gfCNCPoint2[22796] = {X 363.4255, Y 42.5965, Z -3.0000, A 0.000, B 0.000, C 0.000 }
gfCNCPoint2[22797] = {X 362.0806, Y 43.9848, Z -3.0000, A 0.000, B 0.000, C 0.000 }
gfCNCPoint2[22798] = {X 360.6191, Y 45.2499, Z -3.0000, A 0.000, B 0.000, C 0.000 }
gfCNCPoint2[22799] = {X 359.0523, Y 46.3820, Z -3.0000, A 0.000, B 0.000, C 0.000 }
gfCNCPoint2[22800] = {X 357.3923, Y 47.3724, Z -3.0000, A 0.000, B 0.000, C 0.000 }
gfCNCPoint2[22801] = {X 355.4454, Y 48.2565, Z -3.0000, A 0.000, B 0.000, C 0.000 }
gfCNCPoint2[22802] = {X 353.4232, Y 48.9515, Z -3.0000, A 0.000, B 0.000, C 0.000 }
gfCNCPoint2[22803] = {X 351.3441, Y 49.4512, Z -3.0000, A 0.000, B 0.000, C 0.000 }
gfCNCPoint2[22804] = {X 349.2270, Y 49.7510, Z -3.0000, A 0.000, B 0.000, C 0.000 }
gfCNCPoint2[22805] = {X 347.0909, Y 49.8483, Z -3.0000, A 0.000, B 0.000, C 0.000 }
gfCNCPoint2[22806] = {X 345.0381, Y 49.8138, Z -3.0000, A 0.000, B 0.000, C 0.000 }
gfCNCPoint2[22807] = {X 342.9961, Y 49.6015, Z -3.0000, A 0.000, B 0.000, C 0.000 }
gfCNCPoint2[22808] = {X 340.9802, Y 49.2128, Z -3.0000, A 0.000, B 0.000, C 0.000 }
gfCNCPoint2[22809] = {X 339.0056, Y 48.6507, Z -3.0000, A 0.000, B 0.000, C 0.000 }
gfCNCPoint2[22810] = {X 337.0871, Y 47.9195, Z -3.0000, A 0.000, B 0.000, C 0.000 }
gfCNCPoint2[22811] = {X 335.2394, Y 47.0246, Z -3.0000, A 0.000, B 0.000, C 0.000 }
gfCNCPoint2[22812] = {X 333.6461, Y 46.0400, Z -3.0000, A 0.000, B 0.000, C 0.000 }
gfCNCPoint2[22813] = {X 332.1356, Y 44.9327, Z -3.0000, A 0.000, B 0.000, C 0.000 }
gfCNCPoint2[22814] = {X 330.7173, Y 43.7094, Z -3.0000, A 0.000, B 0.000, C 0.000 }
gfCNCPoint2[22815] = {X 329.7931, Y 43.7230, Z -3.0000, A 0.000, B 0.000, C 0.000 }
gfCNCPoint2[22816] = {X 328.8887, Y 43.5322, Z -3.0000, A 0.000, B 0.000, C 0.000 }
gfCNCPoint2[22817] = {X 328.0488, Y 43.1465, Z -3.0000, A 0.000, B 0.000, C 0.000 }
gfCNCPoint2[22818] = {X 327.3148, Y 42.5847, Z -3.0000, A 0.000, B 0.000, C 0.000 }
gfCNCPoint2[22819] = {X 326.6925, Y 41.9780, Z -3.0000, A 0.000, B 0.000, C 0.000 }
gfCNCPoint2[22820] = {X 326.0873, Y 41.2331, Z -3.0000, A 0.000, B 0.000, C 0.000 }
gfCNCPoint2[22821] = {X 325.6690, Y 40.3693, Z -3.0000, A 0.000, B 0.000, C 0.000 }
gfCNCPoint2[22822] = {X 325.4597, Y 39.4326, Z -3.0000, A 0.000, B 0.000, C 0.000 }
gfCNCPoint2[22823] = {X 325.4707, Y 38.4730, Z -3.0000, A 0.000, B 0.000, C 0.000 }
gfCNCPoint2[22824] = {X 325.7013, Y 37.5413, Z -3.0000, A 0.000, B 0.000, C 0.000 }
gfCNCPoint2[22825] = {X 326.1392, Y 36.6874, Z -3.0000, A 0.000, B 0.000, C 0.000 }
gfCNCPoint2[22826] = {X 330.3725, Y 30.3577, Z -3.0000, A 0.000, B 0.000, C 0.000 }
gfCNCPoint2[22827] = {X 330.9516, Y 29.6673, Z -3.0000, A 0.000, B 0.000, C 0.000 }
gfCNCPoint2[22828] = {X 331.6658, Y 29.1179, Z -3.0000, A 0.000, B 0.000, C 0.000 }
gfCNCPoint2[22829] = {X 332.4815, Y 28.7351, Z -3.0000, A 0.000, B 0.000, C 0.000 }
gfCNCPoint2[22830] = {X 333.3606, Y 28.5370, Z -3.0000, A 0.000, B 0.000, C 0.000 }
gfCNCPoint2[22831] = {X 334.2616, Y 28.5327, Z -3.0000, A 0.000, B 0.000, C 0.000 }
gfCNCPoint2[22832] = {X 335.1425, Y 28.7226, Z -3.0000, A 0.000, B 0.000, C 0.000 }
gfCNCPoint2[22833] = {X 335.9617, Y 29.0978, Z -3.0000, A 0.000, B 0.000, C 0.000 }
gfCNCPoint2[22834] = {X 336.6810, Y 29.6405, Z -3.0000, A 0.000, B 0.000, C 0.000 }
gfCNCPoint2[22835] = {X 337.3163, Y 30.2523, Z -3.0000, A 0.000, B 0.000, C 0.000 }
gfCNCPoint2[22836] = {X 337.8308, Y 30.8659, Z -3.0000, A 0.000, B 0.000, C 0.000 }
gfCNCPoint2[22837] = {X 338.2182, Y 31.5666, Z -3.0000, A 0.000, B 0.000, C 0.000 }
gfCNCPoint2[22838] = {X 338.4642, Y 32.3286, Z -3.0000, A 0.000, B 0.000, C 0.000 }
gfCNCPoint2[22839] = {X 338.5597, Y 33.1236, Z -3.0000, A 0.000, B 0.000, C 0.000 }
gfCNCPoint2[22840] = {X 338.5011, Y 33.9222, Z -3.0000, A 0.000, B 0.000, C 0.000 }
gfCNCPoint2[22841] = {X 339.2995, Y 34.6500, Z -3.0000, A 0.000, B 0.000, C 0.000 }
gfCNCPoint2[22842] = {X 340.1353, Y 35.3347, Z -3.0000, A 0.000, B 0.000, C 0.000 }
gfCNCPoint2[22843] = {X 341.4519, Y 36.1996, Z -3.0000, A 0.000, B 0.000, C 0.000 }
gfCNCPoint2[22844] = {X 342.8804, Y 36.8633, Z -3.0000, A 0.000, B 0.000, C 0.000 }
gfCNCPoint2[22845] = {X 344.3905, Y 37.3116, Z -3.0000, A 0.000, B 0.000, C 0.000 }
gfCNCPoint2[22846] = {X 345.9498, Y 37.5350, Z -3.0000, A 0.000, B 0.000, C 0.000 }
gfCNCPoint2[22847] = {X 347.5251, Y 37.5286, Z -3.0000, A 0.000, B 0.000, C 0.000 }
gfCNCPoint2[22848] = {X 348.7008, Y 37.3905, Z -3.0000, A 0.000, B 0.000, C 0.000 }
gfCNCPoint2[22849] = {X 349.8485, Y 37.1001, Z -3.0000, A 0.000, B 0.000, C 0.000 }
gfCNCPoint2[22850] = {X 350.9485, Y 36.6625, Z -3.0000, A 0.000, B 0.000, C 0.000 }
gfCNCPoint2[22851] = {X 351.9820, Y 36.0851, Z -3.0000, A 0.000, B 0.000, C 0.000 }
gfCNCPoint2[22852] = {X 352.9314, Y 35.3779, Z -3.0000, A 0.000, B 0.000, C 0.000 }
gfCNCPoint2[22853] = {X 354.1005, Y 34.2424, Z -3.0000, A 0.000, B 0.000, C 0.000 }
gfCNCPoint2[22854] = {X 355.1123, Y 32.9647, Z -3.0000, A 0.000, B 0.000, C 0.000 }
gfCNCPoint2[22855] = {X 355.9496, Y 31.5665, Z -3.0000, A 0.000, B 0.000, C 0.000 }
gfCNCPoint2[22856] = {X 356.5983, Y 30.0713, Z -3.0000, A 0.000, B 0.000, C 0.000 }
gfCNCPoint2[22857] = {X 357.0473, Y 28.5046, Z -3.0000, A 0.000, B 0.000, C 0.000 }
gfCNCPoint2[22858] = {X 357.3230, Y 26.8012, Z -3.0000, A 0.000, B 0.000, C 0.000 }
gfCNCPoint2[22859] = {X 357.4354, Y 25.0793, Z -3.0000, A 0.000, B 0.000, C 0.000 }
gfCNCPoint2[22860] = {X 357.3833, Y 23.3545, Z -3.0000, A 0.000, B 0.000, C 0.000 }
gfCNCPoint2[22861] = {X 357.1672, Y 21.6425, Z -3.0000, A 0.000, B 0.000, C 0.000 }
gfCNCPoint2[22862] = {X 356.8264, Y 20.1740, Z -3.0000, A 0.000, B 0.000, C 0.000 }
gfCNCPoint2[22863] = {X 356.3065, Y 18.7588, Z -3.0000, A 0.000, B 0.000, C 0.000 }
gfCNCPoint2[22864] = {X 355.6155, Y 17.4189, Z -3.0000, A 0.000, B 0.000, C 0.000 }
gfCNCPoint2[22865] = {X 354.7641, Y 16.1748, Z -3.0000, A 0.000, B 0.000, C 0.000 }
gfCNCPoint2[22866] = {X 353.8628, Y 15.1697, Z -3.0000, A 0.000, B 0.000, C 0.000 }
gfCNCPoint2[22867] = {X 352.8268, Y 14.3041, Z -3.0000, A 0.000, B 0.000, C 0.000 }
gfCNCPoint2[22868] = {X 351.6776, Y 13.5959, Z -3.0000, A 0.000, B 0.000, C 0.000 }
gfCNCPoint2[22869] = {X 350.4387, Y 13.0595, Z -3.0000, A 0.000, B 0.000, C 0.000 }
gfCNCPoint2[22870] = {X 349.1358, Y 12.7062, Z -3.0000, A 0.000, B 0.000, C 0.000 }
gfCNCPoint2[22871] = {X 347.5974, Y 12.5009, Z -3.0000, A 0.000, B 0.000, C 0.000 }
gfCNCPoint2[22872] = {X 346.0456, Y 12.4729, Z -3.0000, A 0.000, B 0.000, C 0.000 }
gfCNCPoint2[22873] = {X 344.5007, Y 12.6227, Z -3.0000, A 0.000, B 0.000, C 0.000 }
gfCNCPoint2[22874] = {X 342.9832, Y 12.9482, Z -3.0000, A 0.000, B 0.000, C 0.000 }
gfCNCPoint2[22875] = {X 341.5129, Y 13.4452, Z -3.0000, A 0.000, B 0.000, C 0.000 }
gfCNCPoint2[22876] = {X 340.1091, Y 14.1071, Z -3.0000, A 0.000, B 0.000, C 0.000 }
gfCNCPoint2[22877] = {X 338.7902, Y 14.9254, Z -3.0000, A 0.000, B 0.000, C 0.000 }
gfCNCPoint2[22878] = {X 338.7680, Y 15.7568, Z -3.0000, A 0.000, B 0.000, C 0.000 }
gfCNCPoint2[22879] = {X 338.5809, Y 16.5673, Z -3.0000, A 0.000, B 0.000, C 0.000 }
gfCNCPoint2[22880] = {X 338.2362, Y 17.3243, Z -3.0000, A 0.000, B 0.000, C 0.000 }
gfCNCPoint2[22881] = {X 337.7479, Y 17.9976, Z -3.0000, A 0.000, B 0.000, C 0.000 }
gfCNCPoint2[22882] = {X 337.1353, Y 18.5603, Z -3.0000, A 0.000, B 0.000, C 0.000 }
gfCNCPoint2[22883] = {X 336.4209, Y 19.0861, Z -3.0000, A 0.000, B 0.000, C 0.000 }
gfCNCPoint2[22884] = {X 335.6353, Y 19.5283, Z -3.0000, A 0.000, B 0.000, C 0.000 }
gfCNCPoint2[22885] = {X 334.7729, Y 19.7908, Z -3.0000, A 0.000, B 0.000, C 0.000 }
gfCNCPoint2[22886] = {X 333.8742, Y 19.8614, Z -3.0000, A 0.000, B 0.000, C 0.000 }
gfCNCPoint2[22887] = {X 332.9814, Y 19.7367, Z -3.0000, A 0.000, B 0.000, C 0.000 }
gfCNCPoint2[22888] = {X 332.1364, Y 19.4226, Z -3.0000, A 0.000, B 0.000, C 0.000 }
gfCNCPoint2[22889] = {X 331.3789, Y 18.9339, Z -3.0000, A 0.000, B 0.000, C 0.000 }
gfCNCPoint2[22890] = {X 330.7445, Y 18.2934, Z -3.0000, A 0.000, B 0.000, C 0.000 }
gfCNCPoint2[22891] = {X 330.2630, Y 17.5314, Z -3.0000, A 0.000, B 0.000, C 0.000 }
gfCNCPoint2[22892] = {X 326.7381, Y 10.2803, Z -3.0000, A 0.000, B 0.000, C 0.000 }
gfCNCPoint2[22893] = {X 326.4156, Y 9.3505, Z -3.0000, A 0.000, B 0.000, C 0.000 }
gfCNCPoint2[22894] = {X 326.3205, Y 8.3711, Z -3.0000, A 0.000, B 0.000, C 0.000 }
gfCNCPoint2[22895] = {X 326.4581, Y 7.3967, Z -3.0000, A 0.000, B 0.000, C 0.000 }
gfCNCPoint2[22896] = {X 326.8207, Y 6.4819, Z -3.0000, A 0.000, B 0.000, C 0.000 }
gfCNCPoint2[22897] = {X 327.3881, Y 5.6778, Z -3.0000, A 0.000, B 0.000, C 0.000 }
gfCNCPoint2[22898] = {X 328.1285, Y 5.0296, Z -3.0000, A 0.000, B 0.000, C 0.000 }
gfCNCPoint2[22899] = {X 328.7983, Y 4.5709, Z -3.0000, A 0.000, B 0.000, C 0.000 }
gfCNCPoint2[22900] = {X 329.6633, Y 4.1255, Z -3.0000, A 0.000, B 0.000, C 0.000 }
gfCNCPoint2[22901] = {X 330.6082, Y 3.8933, Z -3.0000, A 0.000, B 0.000, C 0.000 }
gfCNCPoint2[22902] = {X 331.5811, Y 3.8868, Z -3.0000, A 0.000, B 0.000, C 0.000 }
gfCNCPoint2[22903] = {X 332.5290, Y 4.1066, Z -3.0000, A 0.000, B 0.000, C 0.000 }
gfCNCPoint2[22904] = {X 334.0387, Y 3.2602, Z -3.0000, A 0.000, B 0.000, C 0.000 }
gfCNCPoint2[22905] = {X 335.5974, Y 2.5081, Z -3.0000, A 0.000, B 0.000, C 0.000 }
gfCNCPoint2[22906] = {X 337.7207, Y 1.6466, Z -3.0000, A 0.000, B 0.000, C 0.000 }
gfCNCPoint2[22907] = {X 339.9113, Y 0.9746, Z -3.0000, A 0.000, B 0.000, C 0.000 }
gfCNCPoint2[22908] = {X 342.1523, Y 0.4972, Z -3.0000, A 0.000, B 0.000, C 0.000 }
gfCNCPoint2[22909] = {X 344.4266, Y 0.2179, Z -3.0000, A 0.000, B 0.000, C 0.000 }
gfCNCPoint2[22910] = {X 346.7166, Y 0.1391, Z -3.0000, A 0.000, B 0.000, C 0.000 }
gfCNCPoint2[22911] = {X 349.0046, Y 0.2612, Z -3.0000, A 0.000, B 0.000, C 0.000 }
gfCNCPoint2[22912] = {X 351.2732, Y 0.5834, Z -3.0000, A 0.000, B 0.000, C 0.000 }
gfCNCPoint2[22913] = {X 351.5567, Y 0.6360, Z -3.0000, A 0.000, B 0.000, C 0.000 }
gfCNCPoint2[22914] = {X 352.2862, Y -3.2969, Z -3.0000, A 0.000, B 0.000, C 0.000 }
gfCNCPoint2[22915] = {X 351.5421, Y 0.7147, Z -3.0000, A 0.000, B 0.000, C 0.000 }
gfCNCPoint2[22916] = {X 351.8236, Y 0.7669, Z -3.0000, A 0.000, B 0.000, C 0.000 }
gfCNCPoint2[22917] = {X 353.7359, Y 1.2474, Z -3.0000, A 0.000, B 0.000, C 0.000 }
gfCNCPoint2[22918] = {X 355.5941, Y 1.9070, Z -3.0000, A 0.000, B 0.000, C 0.000 }
gfCNCPoint2[22919] = {X 357.3815, Y 2.7397, Z -3.0000, A 0.000, B 0.000, C 0.000 }
gfCNCPoint2[22920] = {X 359.0818, Y 3.7380, Z -3.0000, A 0.000, B 0.000, C 0.000 }
gfCNCPoint2[22921] = {X 360.6799, Y 4.8930, Z -3.0000, A 0.000, B 0.000, C 0.000 }
gfCNCPoint2[22922] = {X 362.1614, Y 6.1942, Z -3.0000, A 0.000, B 0.000, C 0.000 }
gfCNCPoint2[22923] = {X 363.5129, Y 7.6299, Z -3.0000, A 0.000, B 0.000, C 0.000 }
gfCNCPoint2[22924] = {X 364.9659, Y 9.5050, Z -3.0000, A 0.000, B 0.000, C 0.000 }
gfCNCPoint2[22925] = {X 366.2305, Y 11.5119, Z -3.0000, A 0.000, B 0.000, C 0.000 }
gfCNCPoint2[22926] = {X 367.2950, Y 13.6318, Z -3.0000, A 0.000, B 0.000, C 0.000 }
gfCNCPoint2[22927] = {X 368.1493, Y 15.8448, Z -3.0000, A 0.000, B 0.000, C 0.000 }
gfCNCPoint2[22928] = {X 368.7853, Y 18.1301, Z -3.0000, A 0.000, B 0.000, C 0.000 }
gfCNCPoint2[22929] = {X 369.2628, Y 20.7447, Z -3.0000, A 0.000, B 0.000, C 0.000 }
gfCNCPoint2[22930] = {X 369.5173, Y 23.3903, Z -3.0000, A 0.000, B 0.000, C 0.000 }
gfCNCPoint2[22931] = {X 369.5471, Y 26.0480, Z -3.0000, A 0.000, B 0.000, C 0.000 }
gfCNCPoint2[22932] = {X 369.3519, Y 28.6987, Z -3.0000, A 0.000, B 0.000, C 0.000 }
gfCNCPoint2[22933] = {X 368.9331, Y 31.3234, Z -3.0000, A 0.000, B 0.000, C 0.000 }
gfCNCPoint2[22934] = {X 368.4143, Y 33.4074, Z -3.0000, A 0.000, B 0.000, C 0.000 }
gfCNCPoint2[22935] = {X 367.7134, Y 35.4375, Z -3.0000, A 0.000, B 0.000, C 0.000 }
gfCNCPoint2[22936] = {X 366.8358, Y 37.3977, Z -3.0000, A 0.000, B 0.000, C 0.000 }
gfCNCPoint2[22937] = {X 365.7884, Y 39.2726, Z -3.0000, A 0.000, B 0.000, C 0.000 }
gfCNCPoint2[22938] = {X 364.5794, Y 41.0477, Z -3.0000, A 0.000, B 0.000, C 0.000 }
gfCNCPoint2[22939] = {X 363.3659, Y 42.5431, Z -3.0000, A 0.000, B 0.000, C 0.000 }
gfCNCPoint2[22940] = {X 362.0260, Y 43.9264, Z -3.0000, A 0.000, B 0.000, C 0.000 }
gfCNCPoint2[22941] = {X 360.5699, Y 45.1869, Z -3.0000, A 0.000, B 0.000, C 0.000 }
gfCNCPoint2[22942] = {X 359.0089, Y 46.3148, Z -3.0000, A 0.000, B 0.000, C 0.000 }
gfCNCPoint2[22943] = {X 357.3551, Y 47.3015, Z -3.0000, A 0.000, B 0.000, C 0.000 }
gfCNCPoint2[22944] = {X 355.4150, Y 48.1825, Z -3.0000, A 0.000, B 0.000, C 0.000 }
gfCNCPoint2[22945] = {X 353.3999, Y 48.8750, Z -3.0000, A 0.000, B 0.000, C 0.000 }
gfCNCPoint2[22946] = {X 351.3281, Y 49.3728, Z -3.0000, A 0.000, B 0.000, C 0.000 }
gfCNCPoint2[22947] = {X 349.2184, Y 49.6715, Z -3.0000, A 0.000, B 0.000, C 0.000 }
gfCNCPoint2[22948] = {X 347.0899, Y 49.7683, Z -3.0000, A 0.000, B 0.000, C 0.000 }
gfCNCPoint2[22949] = {X 345.0440, Y 49.7340, Z -3.0000, A 0.000, B 0.000, C 0.000 }
gfCNCPoint2[22950] = {X 343.0088, Y 49.5225, Z -3.0000, A 0.000, B 0.000, C 0.000 }
gfCNCPoint2[22951] = {X 340.9996, Y 49.1352, Z -3.0000, A 0.000, B 0.000, C 0.000 }
gfCNCPoint2[22952] = {X 339.0316, Y 48.5751, Z -3.0000, A 0.000, B 0.000, C 0.000 }
gfCNCPoint2[22953] = {X 337.1196, Y 47.8464, Z -3.0000, A 0.000, B 0.000, C 0.000 }
gfCNCPoint2[22954] = {X 335.2780, Y 46.9545, Z -3.0000, A 0.000, B 0.000, C 0.000 }
gfCNCPoint2[22955] = {X 333.6799, Y 45.9664, Z -3.0000, A 0.000, B 0.000, C 0.000 }
gfCNCPoint2[22956] = {X 332.1655, Y 44.8542, Z -3.0000, A 0.000, B 0.000, C 0.000 }
gfCNCPoint2[22957] = {X 330.7443, Y 43.6252, Z -3.0000, A 0.000, B 0.000, C 0.000 }
gfCNCPoint2[22958] = {X 329.8287, Y 43.6460, Z -3.0000, A 0.000, B 0.000, C 0.000 }
gfCNCPoint2[22959] = {X 328.9316, Y 43.4621, Z -3.0000, A 0.000, B 0.000, C 0.000 }
gfCNCPoint2[22960] = {X 328.0980, Y 43.0827, Z -3.0000, A 0.000, B 0.000, C 0.000 }
gfCNCPoint2[22961] = {X 327.3701, Y 42.5270, Z -3.0000, A 0.000, B 0.000, C 0.000 }
gfCNCPoint2[22962] = {X 326.7483, Y 41.9207, Z -3.0000, A 0.000, B 0.000, C 0.000 }
gfCNCPoint2[22963] = {X 326.1548, Y 41.1901, Z -3.0000, A 0.000, B 0.000, C 0.000 }
gfCNCPoint2[22964] = {X 325.7445, Y 40.3430, Z -3.0000, A 0.000, B 0.000, C 0.000 }
gfCNCPoint2[22965] = {X 325.5393, Y 39.4243, Z -3.0000, A 0.000, B 0.000, C 0.000 }
gfCNCPoint2[22966] = {X 325.5500, Y 38.4831, Z -3.0000, A 0.000, B 0.000, C 0.000 }
gfCNCPoint2[22967] = {X 325.7762, Y 37.5694, Z -3.0000, A 0.000, B 0.000, C 0.000 }
gfCNCPoint2[22968] = {X 326.2057, Y 36.7318, Z -3.0000, A 0.000, B 0.000, C 0.000 }
gfCNCPoint2[22969] = {X 330.4390, Y 30.4021, Z -3.0000, A 0.000, B 0.000, C 0.000 }
gfCNCPoint2[22970] = {X 331.0069, Y 29.7251, Z -3.0000, A 0.000, B 0.000, C 0.000 }
gfCNCPoint2[22971] = {X 331.7073, Y 29.1862, Z -3.0000, A 0.000, B 0.000, C 0.000 }
gfCNCPoint2[22972] = {X 332.5073, Y 28.8108, Z -3.0000, A 0.000, B 0.000, C 0.000 }
gfCNCPoint2[22973] = {X 333.3694, Y 28.6165, Z -3.0000, A 0.000, B 0.000, C 0.000 }
gfCNCPoint2[22974] = {X 334.2530, Y 28.6123, Z -3.0000, A 0.000, B 0.000, C 0.000 }
gfCNCPoint2[22975] = {X 335.1169, Y 28.7985, Z -3.0000, A 0.000, B 0.000, C 0.000 }
gfCNCPoint2[22976] = {X 335.9204, Y 29.1663, Z -3.0000, A 0.000, B 0.000, C 0.000 }
gfCNCPoint2[22977] = {X 336.6259, Y 29.6985, Z -3.0000, A 0.000, B 0.000, C 0.000 }
gfCNCPoint2[22978] = {X 337.2602, Y 30.3094, Z -3.0000, A 0.000, B 0.000, C 0.000 }
gfCNCPoint2[22979] = {X 337.7696, Y 30.9181, Z -3.0000, A 0.000, B 0.000, C 0.000 }
gfCNCPoint2[22980] = {X 338.1515, Y 31.6139, Z -3.0000, A 0.000, B 0.000, C 0.000 }
gfCNCPoint2[22981] = {X 338.3914, Y 32.3705, Z -3.0000, A 0.000, B 0.000, C 0.000 }
gfCNCPoint2[22982] = {X 338.4804, Y 33.1593, Z -3.0000, A 0.000, B 0.000, C 0.000 }
gfCNCPoint2[22983] = {X 338.4149, Y 33.9503, Z -3.0000, A 0.000, B 0.000, C 0.000 }
gfCNCPoint2[22984] = {X 339.2312, Y 34.6967, Z -3.0000, A 0.000, B 0.000, C 0.000 }
gfCNCPoint2[22985] = {X 340.0864, Y 35.3980, Z -3.0000, A 0.000, B 0.000, C 0.000 }
gfCNCPoint2[22986] = {X 341.4126, Y 36.2693, Z -3.0000, A 0.000, B 0.000, C 0.000 }
gfCNCPoint2[22987] = {X 342.8516, Y 36.9379, Z -3.0000, A 0.000, B 0.000, C 0.000 }
gfCNCPoint2[22988] = {X 344.3727, Y 37.3896, Z -3.0000, A 0.000, B 0.000, C 0.000 }
gfCNCPoint2[22989] = {X 345.9434, Y 37.6147, Z -3.0000, A 0.000, B 0.000, C 0.000 }
gfCNCPoint2[22990] = {X 347.5302, Y 37.6085, Z -3.0000, A 0.000, B 0.000, C 0.000 }
gfCNCPoint2[22991] = {X 348.7161, Y 37.4690, Z -3.0000, A 0.000, B 0.000, C 0.000 }
gfCNCPoint2[22992] = {X 349.8737, Y 37.1760, Z -3.0000, A 0.000, B 0.000, C 0.000 }
gfCNCPoint2[22993] = {X 350.9832, Y 36.7345, Z -3.0000, A 0.000, B 0.000, C 0.000 }
gfCNCPoint2[22994] = {X 352.0257, Y 36.1521, Z -3.0000, A 0.000, B 0.000, C 0.000 }
gfCNCPoint2[22995] = {X 352.9832, Y 35.4388, Z -3.0000, A 0.000, B 0.000, C 0.000 }
gfCNCPoint2[22996] = {X 354.1599, Y 34.2960, Z -3.0000, A 0.000, B 0.000, C 0.000 }
gfCNCPoint2[22997] = {X 355.1782, Y 33.0101, Z -3.0000, A 0.000, B 0.000, C 0.000 }
gfCNCPoint2[22998] = {X 356.0208, Y 31.6029, Z -3.0000, A 0.000, B 0.000, C 0.000 }
gfCNCPoint2[22999] = {X 356.6736, Y 30.0982, Z -3.0000, A 0.000, B 0.000, C 0.000 }
gfCNCPoint2[23000] = {X 357.1255, Y 28.5214, Z -3.0000, A 0.000, B 0.000, C 0.000 }
gfCNCPoint2[23001] = {X 357.4025, Y 26.8104, Z -3.0000, A 0.000, B 0.000, C 0.000 }
gfCNCPoint2[23002] = {X 357.5154, Y 25.0808, Z -3.0000, A 0.000, B 0.000, C 0.000 }
gfCNCPoint2[23003] = {X 357.4630, Y 23.3484, Z -3.0000, A 0.000, B 0.000, C 0.000 }
gfCNCPoint2[23004] = {X 357.2460, Y 21.6288, Z -3.0000, A 0.000, B 0.000, C 0.000 }
gfCNCPoint2[23005] = {X 356.9029, Y 20.1507, Z -3.0000, A 0.000, B 0.000, C 0.000 }
gfCNCPoint2[23006] = {X 356.3797, Y 18.7264, Z -3.0000, A 0.000, B 0.000, C 0.000 }
gfCNCPoint2[23007] = {X 355.6842, Y 17.3778, Z -3.0000, A 0.000, B 0.000, C 0.000 }
gfCNCPoint2[23008] = {X 354.8272, Y 16.1256, Z -3.0000, A 0.000, B 0.000, C 0.000 }
gfCNCPoint2[23009] = {X 353.9182, Y 15.1120, Z -3.0000, A 0.000, B 0.000, C 0.000 }
gfCNCPoint2[23010] = {X 352.8735, Y 14.2391, Z -3.0000, A 0.000, B 0.000, C 0.000 }
gfCNCPoint2[23011] = {X 351.7144, Y 13.5249, Z -3.0000, A 0.000, B 0.000, C 0.000 }
gfCNCPoint2[23012] = {X 350.4650, Y 12.9840, Z -3.0000, A 0.000, B 0.000, C 0.000 }
gfCNCPoint2[23013] = {X 349.1511, Y 12.6277, Z -3.0000, A 0.000, B 0.000, C 0.000 }
gfCNCPoint2[23014] = {X 347.5971, Y 12.4206, Z -3.0000, A 0.000, B 0.000, C 0.000 }
gfCNCPoint2[23015] = {X 346.0297, Y 12.3935, Z -3.0000, A 0.000, B 0.000, C 0.000 }
gfCNCPoint2[23016] = {X 344.4695, Y 12.5466, Z -3.0000, A 0.000, B 0.000, C 0.000 }
gfCNCPoint2[23017] = {X 342.9373, Y 12.8779, Z -3.0000, A 0.000, B 0.000, C 0.000 }
gfCNCPoint2[23018] = {X 341.4532, Y 13.3830, Z -3.0000, A 0.000, B 0.000, C 0.000 }
gfCNCPoint2[23019] = {X 340.0371, Y 14.0553, Z -3.0000, A 0.000, B 0.000, C 0.000 }
gfCNCPoint2[23020] = {X 338.7075, Y 14.8858, Z -3.0000, A 0.000, B 0.000, C 0.000 }
gfCNCPoint2[23021] = {X 338.7152, Y 15.0050, Z -3.0000, A 0.000, B 0.000, C 0.000 }
gfCNCPoint2[23022] = {X 338.6808, Y 15.8053, Z -3.0000, A 0.000, B 0.000, C 0.000 }
gfCNCPoint2[23023] = {X 338.4907, Y 16.5835, Z -3.0000, A 0.000, B 0.000, C 0.000 }
gfCNCPoint2[23024] = {X 338.1521, Y 17.3095, Z -3.0000, A 0.000, B 0.000, C 0.000 }
gfCNCPoint2[23025] = {X 337.6783, Y 17.9554, Z -3.0000, A 0.000, B 0.000, C 0.000 }
gfCNCPoint2[23026] = {X 337.0874, Y 18.4963, Z -3.0000, A 0.000, B 0.000, C 0.000 }
gfCNCPoint2[23027] = {X 336.3744, Y 19.0211, Z -3.0000, A 0.000, B 0.000, C 0.000 }
gfCNCPoint2[23028] = {X 335.6039, Y 19.4547, Z -3.0000, A 0.000, B 0.000, C 0.000 }
gfCNCPoint2[23029] = {X 334.7580, Y 19.7122, Z -3.0000, A 0.000, B 0.000, C 0.000 }
gfCNCPoint2[23030] = {X 333.8766, Y 19.7814, Z -3.0000, A 0.000, B 0.000, C 0.000 }
gfCNCPoint2[23031] = {X 333.0010, Y 19.6592, Z -3.0000, A 0.000, B 0.000, C 0.000 }
gfCNCPoint2[23032] = {X 332.1722, Y 19.3511, Z -3.0000, A 0.000, B 0.000, C 0.000 }
gfCNCPoint2[23033] = {X 331.4293, Y 18.8718, Z -3.0000, A 0.000, B 0.000, C 0.000 }
gfCNCPoint2[23034] = {X 330.8071, Y 18.2436, Z -3.0000, A 0.000, B 0.000, C 0.000 }
gfCNCPoint2[23035] = {X 330.3348, Y 17.4962, Z -3.0000, A 0.000, B 0.000, C 0.000 }
gfCNCPoint2[23036] = {X 326.8100, Y 10.2453, Z -3.0000, A 0.000, B 0.000, C 0.000 }
gfCNCPoint2[23037] = {X 326.4937, Y 9.3334, Z -3.0000, A 0.000, B 0.000, C 0.000 }
gfCNCPoint2[23038] = {X 326.4004, Y 8.3728, Z -3.0000, A 0.000, B 0.000, C 0.000 }
gfCNCPoint2[23039] = {X 326.5354, Y 7.4171, Z -3.0000, A 0.000, B 0.000, C 0.000 }
gfCNCPoint2[23040] = {X 326.8911, Y 6.5199, Z -3.0000, A 0.000, B 0.000, C 0.000 }
gfCNCPoint2[23041] = {X 327.4476, Y 5.7314, Z -3.0000, A 0.000, B 0.000, C 0.000 }
gfCNCPoint2[23042] = {X 328.1737, Y 5.0956, Z -3.0000, A 0.000, B 0.000, C 0.000 }
gfCNCPoint2[23043] = {X 328.8432, Y 4.6371, Z -3.0000, A 0.000, B 0.000, C 0.000 }
gfCNCPoint2[23044] = {X 329.7005, Y 4.1971, Z -3.0000, A 0.000, B 0.000, C 0.000 }
gfCNCPoint2[23045] = {X 330.6370, Y 3.9704, Z -3.0000, A 0.000, B 0.000, C 0.000 }
gfCNCPoint2[23046] = {X 331.6006, Y 3.9696, Z -3.0000, A 0.000, B 0.000, C 0.000 }
gfCNCPoint2[23047] = {X 332.5375, Y 4.1949, Z -3.0000, A 0.000, B 0.000, C 0.000 }
gfCNCPoint2[23048] = {X 334.0589, Y 3.3399, Z -3.0000, A 0.000, B 0.000, C 0.000 }
gfCNCPoint2[23049] = {X 335.6304, Y 2.5810, Z -3.0000, A 0.000, B 0.000, C 0.000 }
gfCNCPoint2[23050] = {X 337.7472, Y 1.7221, Z -3.0000, A 0.000, B 0.000, C 0.000 }
gfCNCPoint2[23051] = {X 339.9311, Y 1.0521, Z -3.0000, A 0.000, B 0.000, C 0.000 }
gfCNCPoint2[23052] = {X 342.1653, Y 0.5761, Z -3.0000, A 0.000, B 0.000, C 0.000 }
gfCNCPoint2[23053] = {X 344.4327, Y 0.2977, Z -3.0000, A 0.000, B 0.000, C 0.000 }
gfCNCPoint2[23054] = {X 346.7157, Y 0.2191, Z -3.0000, A 0.000, B 0.000, C 0.000 }
gfCNCPoint2[23055] = {X 348.9968, Y 0.3409, Z -3.0000, A 0.000, B 0.000, C 0.000 }
gfCNCPoint2[23056] = {X 351.2585, Y 0.6621, Z -3.0000, A 0.000, B 0.000, C 0.000 }
gfCNCPoint2[23057] = {X 351.5421, Y 0.7147, Z -3.0000, A 0.000, B 0.000, C 0.000 }
gfCNCPoint2[23058] = {X 352.2716, Y -3.2182, Z -3.0000, A 0.000, B 0.000, C 0.000 }
gfCNCPoint2[23059] = {X 351.5276, Y 0.7933, Z -3.0000, A 0.000, B 0.000, C 0.000 }
gfCNCPoint2[23060] = {X 351.8084, Y 0.8454, Z -3.0000, A 0.000, B 0.000, C 0.000 }
gfCNCPoint2[23061] = {X 353.7133, Y 1.3241, Z -3.0000, A 0.000, B 0.000, C 0.000 }
gfCNCPoint2[23062] = {X 355.5642, Y 1.9812, Z -3.0000, A 0.000, B 0.000, C 0.000 }
gfCNCPoint2[23063] = {X 357.3446, Y 2.8107, Z -3.0000, A 0.000, B 0.000, C 0.000 }
gfCNCPoint2[23064] = {X 359.0383, Y 3.8052, Z -3.0000, A 0.000, B 0.000, C 0.000 }
gfCNCPoint2[23065] = {X 360.6302, Y 4.9557, Z -3.0000, A 0.000, B 0.000, C 0.000 }
gfCNCPoint2[23066] = {X 362.1059, Y 6.2518, Z -3.0000, A 0.000, B 0.000, C 0.000 }
gfCNCPoint2[23067] = {X 363.4521, Y 7.6820, Z -3.0000, A 0.000, B 0.000, C 0.000 }
gfCNCPoint2[23068] = {X 364.9004, Y 9.5509, Z -3.0000, A 0.000, B 0.000, C 0.000 }
gfCNCPoint2[23069] = {X 366.1609, Y 11.5513, Z -3.0000, A 0.000, B 0.000, C 0.000 }
gfCNCPoint2[23070] = {X 367.2218, Y 13.6642, Z -3.0000, A 0.000, B 0.000, C 0.000 }
gfCNCPoint2[23071] = {X 368.0733, Y 15.8700, Z -3.0000, A 0.000, B 0.000, C 0.000 }
gfCNCPoint2[23072] = {X 368.7073, Y 18.1478, Z -3.0000, A 0.000, B 0.000, C 0.000 }
gfCNCPoint2[23073] = {X 369.1835, Y 20.7557, Z -3.0000, A 0.000, B 0.000, C 0.000 }
gfCNCPoint2[23074] = {X 369.4374, Y 23.3946, Z -3.0000, A 0.000, B 0.000, C 0.000 }
gfCNCPoint2[23075] = {X 369.4671, Y 26.0455, Z -3.0000, A 0.000, B 0.000, C 0.000 }
gfCNCPoint2[23076] = {X 369.2724, Y 28.6894, Z -3.0000, A 0.000, B 0.000, C 0.000 }
gfCNCPoint2[23077] = {X 368.8548, Y 31.3074, Z -3.0000, A 0.000, B 0.000, C 0.000 }
gfCNCPoint2[23078] = {X 368.3377, Y 33.3847, Z -3.0000, A 0.000, B 0.000, C 0.000 }
gfCNCPoint2[23079] = {X 367.6390, Y 35.4081, Z -3.0000, A 0.000, B 0.000, C 0.000 }
gfCNCPoint2[23080] = {X 366.7643, Y 37.3618, Z -3.0000, A 0.000, B 0.000, C 0.000 }
gfCNCPoint2[23081] = {X 365.7203, Y 39.2306, Z -3.0000, A 0.000, B 0.000, C 0.000 }
gfCNCPoint2[23082] = {X 364.5152, Y 40.9999, Z -3.0000, A 0.000, B 0.000, C 0.000 }
gfCNCPoint2[23083] = {X 363.3063, Y 42.4898, Z -3.0000, A 0.000, B 0.000, C 0.000 }
gfCNCPoint2[23084] = {X 361.9713, Y 43.8680, Z -3.0000, A 0.000, B 0.000, C 0.000 }
gfCNCPoint2[23085] = {X 360.5207, Y 45.1238, Z -3.0000, A 0.000, B 0.000, C 0.000 }
gfCNCPoint2[23086] = {X 358.9655, Y 46.2476, Z -3.0000, A 0.000, B 0.000, C 0.000 }
gfCNCPoint2[23087] = {X 357.3179, Y 47.2307, Z -3.0000, A 0.000, B 0.000, C 0.000 }
gfCNCPoint2[23088] = {X 355.3846, Y 48.1085, Z -3.0000, A 0.000, B 0.000, C 0.000 }
gfCNCPoint2[23089] = {X 353.3766, Y 48.7984, Z -3.0000, A 0.000, B 0.000, C 0.000 }
gfCNCPoint2[23090] = {X 351.3122, Y 49.2944, Z -3.0000, A 0.000, B 0.000, C 0.000 }
gfCNCPoint2[23091] = {X 349.2099, Y 49.5919, Z -3.0000, A 0.000, B 0.000, C 0.000 }
gfCNCPoint2[23092] = {X 347.0889, Y 49.6883, Z -3.0000, A 0.000, B 0.000, C 0.000 }
gfCNCPoint2[23093] = {X 345.0499, Y 49.6542, Z -3.0000, A 0.000, B 0.000, C 0.000 }
gfCNCPoint2[23094] = {X 343.0216, Y 49.4435, Z -3.0000, A 0.000, B 0.000, C 0.000 }
gfCNCPoint2[23095] = {X 341.0191, Y 49.0576, Z -3.0000, A 0.000, B 0.000, C 0.000 }
gfCNCPoint2[23096] = {X 339.0577, Y 48.4994, Z -3.0000, A 0.000, B 0.000, C 0.000 }
gfCNCPoint2[23097] = {X 337.1521, Y 47.7733, Z -3.0000, A 0.000, B 0.000, C 0.000 }
gfCNCPoint2[23098] = {X 335.3167, Y 46.8845, Z -3.0000, A 0.000, B 0.000, C 0.000 }
gfCNCPoint2[23099] = {X 333.7137, Y 45.8926, Z -3.0000, A 0.000, B 0.000, C 0.000 }
gfCNCPoint2[23100] = {X 332.1953, Y 44.7756, Z -3.0000, A 0.000, B 0.000, C 0.000 }
gfCNCPoint2[23101] = {X 330.7711, Y 43.5406, Z -3.0000, A 0.000, B 0.000, C 0.000 }
gfCNCPoint2[23102] = {X 329.8559, Y 43.5681, Z -3.0000, A 0.000, B 0.000, C 0.000 }
gfCNCPoint2[23103] = {X 328.9583, Y 43.3867, Z -3.0000, A 0.000, B 0.000, C 0.000 }
gfCNCPoint2[23104] = {X 328.1256, Y 43.0059, Z -3.0000, A 0.000, B 0.000, C 0.000 }
gfCNCPoint2[23105] = {X 327.4012, Y 42.4458, Z -3.0000, A 0.000, B 0.000, C 0.000 }
gfCNCPoint2[23106] = {X 326.8042, Y 41.8634, Z -3.0000, A 0.000, B 0.000, C 0.000 }
gfCNCPoint2[23107] = {X 326.2223, Y 41.1472, Z -3.0000, A 0.000, B 0.000, C 0.000 }
gfCNCPoint2[23108] = {X 325.8201, Y 40.3166, Z -3.0000, A 0.000, B 0.000, C 0.000 }
gfCNCPoint2[23109] = {X 325.6189, Y 39.4160, Z -3.0000, A 0.000, B 0.000, C 0.000 }
gfCNCPoint2[23110] = {X 325.6294, Y 38.4932, Z -3.0000, A 0.000, B 0.000, C 0.000 }
gfCNCPoint2[23111] = {X 325.8511, Y 37.5974, Z -3.0000, A 0.000, B 0.000, C 0.000 }
gfCNCPoint2[23112] = {X 326.2722, Y 36.7763, Z -3.0000, A 0.000, B 0.000, C 0.000 }
gfCNCPoint2[23113] = {X 330.5290, Y 30.4119, Z -3.0000, A 0.000, B 0.000, C 0.000 }
gfCNCPoint2[23114] = {X 331.0932, Y 29.7535, Z -3.0000, A 0.000, B 0.000, C 0.000 }
gfCNCPoint2[23115] = {X 331.7861, Y 29.2322, Z -3.0000, A 0.000, B 0.000, C 0.000 }
gfCNCPoint2[23116] = {X 332.5750, Y 28.8724, Z -3.0000, A 0.000, B 0.000, C 0.000 }
gfCNCPoint2[23117] = {X 333.4230, Y 28.6911, Z -3.0000, A 0.000, B 0.000, C 0.000 }
gfCNCPoint2[23118] = {X 334.2900, Y 28.6968, Z -3.0000, A 0.000, B 0.000, C 0.000 }
gfCNCPoint2[23119] = {X 335.1355, Y 28.8892, Z -3.0000, A 0.000, B 0.000, C 0.000 }
gfCNCPoint2[23120] = {X 335.9197, Y 29.2593, Z -3.0000, A 0.000, B 0.000, C 0.000 }
gfCNCPoint2[23121] = {X 336.6057, Y 29.7897, Z -3.0000, A 0.000, B 0.000, C 0.000 }
gfCNCPoint2[23122] = {X 337.2041, Y 30.3665, Z -3.0000, A 0.000, B 0.000, C 0.000 }
gfCNCPoint2[23123] = {X 337.7083, Y 30.9703, Z -3.0000, A 0.000, B 0.000, C 0.000 }
gfCNCPoint2[23124] = {X 338.0846, Y 31.6611, Z -3.0000, A 0.000, B 0.000, C 0.000 }
gfCNCPoint2[23125] = {X 338.3184, Y 32.4122, Z -3.0000, A 0.000, B 0.000, C 0.000 }
gfCNCPoint2[23126] = {X 338.4007, Y 33.1945, Z -3.0000, A 0.000, B 0.000, C 0.000 }
gfCNCPoint2[23127] = {X 338.3283, Y 33.9779, Z -3.0000, A 0.000, B 0.000, C 0.000 }
gfCNCPoint2[23128] = {X 339.1626, Y 34.7431, Z -3.0000, A 0.000, B 0.000, C 0.000 }
gfCNCPoint2[23129] = {X 340.0375, Y 35.4613, Z -3.0000, A 0.000, B 0.000, C 0.000 }
gfCNCPoint2[23130] = {X 341.2955, Y 36.2947, Z -3.0000, A 0.000, B 0.000, C 0.000 }
gfCNCPoint2[23131] = {X 342.6562, Y 36.9469, Z -3.0000, A 0.000, B 0.000, C 0.000 }
gfCNCPoint2[23132] = {X 344.0938, Y 37.4056, Z -3.0000, A 0.000, B 0.000, C 0.000 }
gfCNCPoint2[23133] = {X 345.5808, Y 37.6621, Z -3.0000, A 0.000, B 0.000, C 0.000 }
gfCNCPoint2[23134] = {X 347.0889, Y 37.7114, Z -3.0000, A 0.000, B 0.000, C 0.000 }
gfCNCPoint2[23135] = {X 347.5343, Y 37.6884, Z -3.0000, A 0.000, B 0.000, C 0.000 }
gfCNCPoint2[23136] = {X 348.7306, Y 37.5476, Z -3.0000, A 0.000, B 0.000, C 0.000 }
gfCNCPoint2[23137] = {X 349.8984, Y 37.2521, Z -3.0000, A 0.000, B 0.000, C 0.000 }
gfCNCPoint2[23138] = {X 351.0176, Y 36.8068, Z -3.0000, A 0.000, B 0.000, C 0.000 }
gfCNCPoint2[23139] = {X 352.0692, Y 36.2193, Z -3.0000, A 0.000, B 0.000, C 0.000 }
gfCNCPoint2[23140] = {X 353.0351, Y 35.4997, Z -3.0000, A 0.000, B 0.000, C 0.000 }
gfCNCPoint2[23141] = {X 354.2193, Y 34.3496, Z -3.0000, A 0.000, B 0.000, C 0.000 }
gfCNCPoint2[23142] = {X 355.2440, Y 33.0555, Z -3.0000, A 0.000, B 0.000, C 0.000 }
gfCNCPoint2[23143] = {X 356.0921, Y 31.6393, Z -3.0000, A 0.000, B 0.000, C 0.000 }
gfCNCPoint2[23144] = {X 356.7490, Y 30.1250, Z -3.0000, A 0.000, B 0.000, C 0.000 }
gfCNCPoint2[23145] = {X 357.2037, Y 28.5381, Z -3.0000, A 0.000, B 0.000, C 0.000 }
gfCNCPoint2[23146] = {X 357.4820, Y 26.8196, Z -3.0000, A 0.000, B 0.000, C 0.000 }
gfCNCPoint2[23147] = {X 357.5953, Y 25.0823, Z -3.0000, A 0.000, B 0.000, C 0.000 }
gfCNCPoint2[23148] = {X 357.5428, Y 23.3422, Z -3.0000, A 0.000, B 0.000, C 0.000 }
gfCNCPoint2[23149] = {X 357.3248, Y 21.6150, Z -3.0000, A 0.000, B 0.000, C 0.000 }
gfCNCPoint2[23150] = {X 356.9795, Y 20.1274, Z -3.0000, A 0.000, B 0.000, C 0.000 }
gfCNCPoint2[23151] = {X 356.4528, Y 18.6939, Z -3.0000, A 0.000, B 0.000, C 0.000 }
gfCNCPoint2[23152] = {X 355.7528, Y 17.3367, Z -3.0000, A 0.000, B 0.000, C 0.000 }
gfCNCPoint2[23153] = {X 354.8902, Y 16.0764, Z -3.0000, A 0.000, B 0.000, C 0.000 }
gfCNCPoint2[23154] = {X 353.9736, Y 15.0543, Z -3.0000, A 0.000, B 0.000, C 0.000 }
gfCNCPoint2[23155] = {X 352.9201, Y 14.1741, Z -3.0000, A 0.000, B 0.000, C 0.000 }
gfCNCPoint2[23156] = {X 351.7513, Y 13.4539, Z -3.0000, A 0.000, B 0.000, C 0.000 }
gfCNCPoint2[23157] = {X 350.4914, Y 12.9085, Z -3.0000, A 0.000, B 0.000, C 0.000 }
gfCNCPoint2[23158] = {X 349.1664, Y 12.5492, Z -3.0000, A 0.000, B 0.000, C 0.000 }
gfCNCPoint2[23159] = {X 347.3712, Y 12.3254, Z -3.0000, A 0.000, B 0.000, C 0.000 }
gfCNCPoint2[23160] = {X 345.5623, Y 12.3401, Z -3.0000, A 0.000, B 0.000, C 0.000 }
gfCNCPoint2[23161] = {X 343.7710, Y 12.5930, Z -3.0000, A 0.000, B 0.000, C 0.000 }
gfCNCPoint2[23162] = {X 342.0287, Y 13.0796, Z -3.0000, A 0.000, B 0.000, C 0.000 }
gfCNCPoint2[23163] = {X 340.3656, Y 13.7914, Z -3.0000, A 0.000, B 0.000, C 0.000 }
gfCNCPoint2[23164] = {X 338.8108, Y 14.7161, Z -3.0000, A 0.000, B 0.000, C 0.000 }
gfCNCPoint2[23165] = {X 338.7175, Y 14.7809, Z -3.0000, A 0.000, B 0.000, C 0.000 }
gfCNCPoint2[23166] = {X 338.6248, Y 14.8464, Z -3.0000, A 0.000, B 0.000, C 0.000 }
gfCNCPoint2[23167] = {X 338.6379, Y 15.0625, Z -3.0000, A 0.000, B 0.000, C 0.000 }
gfCNCPoint2[23168] = {X 338.5597, Y 16.0351, Z -3.0000, A 0.000, B 0.000, C 0.000 }
gfCNCPoint2[23169] = {X 338.2484, Y 16.9598, Z -3.0000, A 0.000, B 0.000, C 0.000 }
gfCNCPoint2[23170] = {X 337.7225, Y 17.7817, Z -3.0000, A 0.000, B 0.000, C 0.000 }
gfCNCPoint2[23171] = {X 337.0132, Y 18.4517, Z -3.0000, A 0.000, B 0.000, C 0.000 }
gfCNCPoint2[23172] = {X 336.3278, Y 18.9560, Z -3.0000, A 0.000, B 0.000, C 0.000 }
gfCNCPoint2[23173] = {X 335.5713, Y 19.3817, Z -3.0000, A 0.000, B 0.000, C 0.000 }
gfCNCPoint2[23174] = {X 334.7407, Y 19.6341, Z -3.0000, A 0.000, B 0.000, C 0.000 }
gfCNCPoint2[23175] = {X 333.8753, Y 19.7014, Z -3.0000, A 0.000, B 0.000, C 0.000 }
gfCNCPoint2[23176] = {X 333.0157, Y 19.5804, Z -3.0000, A 0.000, B 0.000, C 0.000 }
gfCNCPoint2[23177] = {X 332.2025, Y 19.2768, Z -3.0000, A 0.000, B 0.000, C 0.000 }
gfCNCPoint2[23178] = {X 331.4739, Y 18.8049, Z -3.0000, A 0.000, B 0.000, C 0.000 }
gfCNCPoint2[23179] = {X 330.8643, Y 18.1870, Z -3.0000, A 0.000, B 0.000, C 0.000 }
gfCNCPoint2[23180] = {X 330.4023, Y 17.4521, Z -3.0000, A 0.000, B 0.000, C 0.000 }
gfCNCPoint2[23181] = {X 326.8820, Y 10.2103, Z -3.0000, A 0.000, B 0.000, C 0.000 }
gfCNCPoint2[23182] = {X 326.5719, Y 9.3163, Z -3.0000, A 0.000, B 0.000, C 0.000 }
gfCNCPoint2[23183] = {X 326.4804, Y 8.3746, Z -3.0000, A 0.000, B 0.000, C 0.000 }
gfCNCPoint2[23184] = {X 326.6127, Y 7.4376, Z -3.0000, A 0.000, B 0.000, C 0.000 }
gfCNCPoint2[23185] = {X 326.9614, Y 6.5580, Z -3.0000, A 0.000, B 0.000, C 0.000 }
gfCNCPoint2[23186] = {X 327.5070, Y 5.7849, Z -3.0000, A 0.000, B 0.000, C 0.000 }
gfCNCPoint2[23187] = {X 328.2189, Y 5.1616, Z -3.0000, A 0.000, B 0.000, C 0.000 }
gfCNCPoint2[23188] = {X 328.8880, Y 4.7034, Z -3.0000, A 0.000, B 0.000, C 0.000 }
gfCNCPoint2[23189] = {X 329.7043, Y 4.2813, Z -3.0000, A 0.000, B 0.000, C 0.000 }
gfCNCPoint2[23190] = {X 330.5954, Y 4.0567, Z -3.0000, A 0.000, B 0.000, C 0.000 }
gfCNCPoint2[23191] = {X 331.5142, Y 4.0413, Z -3.0000, A 0.000, B 0.000, C 0.000 }
gfCNCPoint2[23192] = {X 332.4122, Y 4.2361, Z -3.0000, A 0.000, B 0.000, C 0.000 }
gfCNCPoint2[23193] = {X 332.5467, Y 4.2827, Z -3.0000, A 0.000, B 0.000, C 0.000 }
gfCNCPoint2[23194] = {X 332.6260, Y 4.2349, Z -3.0000, A 0.000, B 0.000, C 0.000 }
gfCNCPoint2[23195] = {X 332.7055, Y 4.1874, Z -3.0000, A 0.000, B 0.000, C 0.000 }
gfCNCPoint2[23196] = {X 334.1614, Y 3.3767, Z -3.0000, A 0.000, B 0.000, C 0.000 }
gfCNCPoint2[23197] = {X 335.6629, Y 2.6540, Z -3.0000, A 0.000, B 0.000, C 0.000 }
gfCNCPoint2[23198] = {X 336.0092, Y 2.4999, Z -3.0000, A 0.000, B 0.000, C 0.000 }
gfCNCPoint2[23199] = {X 338.0805, Y 1.6918, Z -3.0000, A 0.000, B 0.000, C 0.000 }
gfCNCPoint2[23200] = {X 340.2133, Y 1.0639, Z -3.0000, A 0.000, B 0.000, C 0.000 }
gfCNCPoint2[23201] = {X 342.3920, Y 0.6209, Z -3.0000, A 0.000, B 0.000, C 0.000 }
gfCNCPoint2[23202] = {X 344.6007, Y 0.3658, Z -3.0000, A 0.000, B 0.000, C 0.000 }
gfCNCPoint2[23203] = {X 346.8231, Y 0.3007, Z -3.0000, A 0.000, B 0.000, C 0.000 }
gfCNCPoint2[23204] = {X 349.0429, Y 0.4260, Z -3.0000, A 0.000, B 0.000, C 0.000 }
gfCNCPoint2[23205] = {X 351.2438, Y 0.7407, Z -3.0000, A 0.000, B 0.000, C 0.000 }
gfCNCPoint2[23206] = {X 351.5276, Y 0.7933, Z -3.0000, A 0.000, B 0.000, C 0.000 }
gfCNCPoint2[23207] = {X 352.2716, Y -3.2182, Z -3.0000, A 0.000, B 0.000, C 0.000 }
gfCNCPoint2[23208] = {X 352.2716, Y -3.2182, Z 0.0000, A 0.000, B 0.000, C 0.000 }
gfCNCPoint2[23209] = {X 352.2716, Y -3.2182, Z 11.0000, A 0.000, B 0.000, C 0.000 }
gfCNCPoint2[23210] = {X 606.0427, Y 42.9010, Z 11.0000, A 0.000, B 0.000, C 0.000 }
gfCNCPoint2[23211] = {X 606.0427, Y 42.9010, Z 0.0000, A 0.000, B 0.000, C 0.000 }
gfCNCPoint2[23212] = {X 606.0427, Y 42.9010, Z -3.0000, A 0.000, B 0.000, C 0.000 }
gfCNCPoint2[23213] = {X 603.6965, Y 47.0769, Z -3.0000, A 0.000, B 0.000, C 0.000 }
gfCNCPoint2[23214] = {X 603.6310, Y 47.1894, Z -3.0000, A 0.000, B 0.000, C 0.000 }
gfCNCPoint2[23215] = {X 603.5621, Y 47.2998, Z -3.0000, A 0.000, B 0.000, C 0.000 }
gfCNCPoint2[23216] = {X 603.0357, Y 47.9601, Z -3.0000, A 0.000, B 0.000, C 0.000 }
gfCNCPoint2[23217] = {X 602.3888, Y 48.5030, Z -3.0000, A 0.000, B 0.000, C 0.000 }
gfCNCPoint2[23218] = {X 601.6472, Y 48.9069, Z -3.0000, A 0.000, B 0.000, C 0.000 }
gfCNCPoint2[23219] = {X 600.8403, Y 49.1559, Z -3.0000, A 0.000, B 0.000, C 0.000 }
gfCNCPoint2[23220] = {X 600.0000, Y 49.2400, Z -3.0000, A 0.000, B 0.000, C 0.000 }
gfCNCPoint2[23221] = {X 593.5565, Y 49.2400, Z -3.0000, A 0.000, B 0.000, C 0.000 }
gfCNCPoint2[23222] = {X 592.6130, Y 49.1337, Z -3.0000, A 0.000, B 0.000, C 0.000 }
gfCNCPoint2[23223] = {X 591.7169, Y 48.8201, Z -3.0000, A 0.000, B 0.000, C 0.000 }
gfCNCPoint2[23224] = {X 590.9129, Y 48.3150, Z -3.0000, A 0.000, B 0.000, C 0.000 }
gfCNCPoint2[23225] = {X 590.2416, Y 47.6436, Z -3.0000, A 0.000, B 0.000, C 0.000 }
gfCNCPoint2[23226] = {X 589.7364, Y 46.8397, Z -3.0000, A 0.000, B 0.000, C 0.000 }
gfCNCPoint2[23227] = {X 589.4228, Y 45.9435, Z -3.0000, A 0.000, B 0.000, C 0.000 }
gfCNCPoint2[23228] = {X 589.3165, Y 45.0000, Z -3.0000, A 0.000, B 0.000, C 0.000 }
gfCNCPoint2[23229] = {X 589.3165, Y 44.0648, Z -3.0000, A 0.000, B 0.000, C 0.000 }
gfCNCPoint2[23230] = {X 589.4213, Y 43.1447, Z -3.0000, A 0.000, B 0.000, C 0.000 }
gfCNCPoint2[23231] = {X 589.7213, Y 42.2687, Z -3.0000, A 0.000, B 0.000, C 0.000 }
gfCNCPoint2[23232] = {X 590.2027, Y 41.4777, Z -3.0000, A 0.000, B 0.000, C 0.000 }
gfCNCPoint2[23233] = {X 590.8428, Y 40.8085, Z -3.0000, A 0.000, B 0.000, C 0.000 }
gfCNCPoint2[23234] = {X 590.8432, Y 33.1194, Z -3.0000, A 0.000, B 0.000, C 0.000 }
gfCNCPoint2[23235] = {X 585.3714, Y 46.6218, Z -3.0000, A 0.000, B 0.000, C 0.000 }
gfCNCPoint2[23236] = {X 585.0085, Y 47.3114, Z -3.0000, A 0.000, B 0.000, C 0.000 }
gfCNCPoint2[23237] = {X 584.5255, Y 47.9228, Z -3.0000, A 0.000, B 0.000, C 0.000 }
gfCNCPoint2[23238] = {X 583.9387, Y 48.4356, Z -3.0000, A 0.000, B 0.000, C 0.000 }
gfCNCPoint2[23239] = {X 583.2680, Y 48.8323, Z -3.0000, A 0.000, B 0.000, C 0.000 }
gfCNCPoint2[23240] = {X 582.3418, Y 49.1460, Z -3.0000, A 0.000, B 0.000, C 0.000 }
gfCNCPoint2[23241] = {X 581.3682, Y 49.2391, Z -3.0000, A 0.000, B 0.000, C 0.000 }
gfCNCPoint2[23242] = {X 580.3993, Y 49.1068, Z -3.0000, A 0.000, B 0.000, C 0.000 }
gfCNCPoint2[23243] = {X 579.4864, Y 48.7559, Z -3.0000, A 0.000, B 0.000, C 0.000 }
gfCNCPoint2[23244] = {X 578.6782, Y 48.2052, Z -3.0000, A 0.000, B 0.000, C 0.000 }
gfCNCPoint2[23245] = {X 578.0177, Y 47.4840, Z -3.0000, A 0.000, B 0.000, C 0.000 }
gfCNCPoint2[23246] = {X 577.5400, Y 46.6307, Z -3.0000, A 0.000, B 0.000, C 0.000 }
gfCNCPoint2[23247] = {X 571.9382, Y 32.9329, Z -3.0000, A 0.000, B 0.000, C 0.000 }
gfCNCPoint2[23248] = {X 571.9386, Y 40.8078, Z -3.0000, A 0.000, B 0.000, C 0.000 }
gfCNCPoint2[23249] = {X 571.9705, Y 40.8336, Z -3.0000, A 0.000, B 0.000, C 0.000 }
gfCNCPoint2[23250] = {X 572.5958, Y 41.4920, Z -3.0000, A 0.000, B 0.000, C 0.000 }
gfCNCPoint2[23251] = {X 573.0666, Y 42.2685, Z -3.0000, A 0.000, B 0.000, C 0.000 }
gfCNCPoint2[23252] = {X 573.3613, Y 43.1275, Z -3.0000, A 0.000, B 0.000, C 0.000 }
gfCNCPoint2[23253] = {X 573.4663, Y 44.0294, Z -3.0000, A 0.000, B 0.000, C 0.000 }
gfCNCPoint2[23254] = {X 573.4664, Y 45.0000, Z -3.0000, A 0.000, B 0.000, C 0.000 }
gfCNCPoint2[23255] = {X 573.3601, Y 45.9435, Z -3.0000, A 0.000, B 0.000, C 0.000 }
gfCNCPoint2[23256] = {X 573.0465, Y 46.8397, Z -3.0000, A 0.000, B 0.000, C 0.000 }
gfCNCPoint2[23257] = {X 572.5414, Y 47.6436, Z -3.0000, A 0.000, B 0.000, C 0.000 }
gfCNCPoint2[23258] = {X 571.8700, Y 48.3150, Z -3.0000, A 0.000, B 0.000, C 0.000 }
gfCNCPoint2[23259] = {X 571.0661, Y 48.8201, Z -3.0000, A 0.000, B 0.000, C 0.000 }
gfCNCPoint2[23260] = {X 570.1699, Y 49.1337, Z -3.0000, A 0.000, B 0.000, C 0.000 }
gfCNCPoint2[23261] = {X 569.2264, Y 49.2400, Z -3.0000, A 0.000, B 0.000, C 0.000 }
gfCNCPoint2[23262] = {X 562.4443, Y 49.2400, Z -3.0000, A 0.000, B 0.000, C 0.000 }
gfCNCPoint2[23263] = {X 561.5008, Y 49.1337, Z -3.0000, A 0.000, B 0.000, C 0.000 }
gfCNCPoint2[23264] = {X 560.6046, Y 48.8201, Z -3.0000, A 0.000, B 0.000, C 0.000 }
gfCNCPoint2[23265] = {X 559.8007, Y 48.3150, Z -3.0000, A 0.000, B 0.000, C 0.000 }
gfCNCPoint2[23266] = {X 559.1293, Y 47.6436, Z -3.0000, A 0.000, B 0.000, C 0.000 }
gfCNCPoint2[23267] = {X 558.6242, Y 46.8397, Z -3.0000, A 0.000, B 0.000, C 0.000 }
gfCNCPoint2[23268] = {X 558.3106, Y 45.9435, Z -3.0000, A 0.000, B 0.000, C 0.000 }
gfCNCPoint2[23269] = {X 558.2043, Y 45.0000, Z -3.0000, A 0.000, B 0.000, C 0.000 }
gfCNCPoint2[23270] = {X 558.2043, Y 44.0649, Z -3.0000, A 0.000, B 0.000, C 0.000 }
gfCNCPoint2[23271] = {X 558.3089, Y 43.1444, Z -3.0000, A 0.000, B 0.000, C 0.000 }
gfCNCPoint2[23272] = {X 558.6092, Y 42.2681, Z -3.0000, A 0.000, B 0.000, C 0.000 }
gfCNCPoint2[23273] = {X 559.0913, Y 41.4770, Z -3.0000, A 0.000, B 0.000, C 0.000 }
gfCNCPoint2[23274] = {X 559.7324, Y 40.8083, Z -3.0000, A 0.000, B 0.000, C 0.000 }
gfCNCPoint2[23275] = {X 559.7324, Y 9.1934, Z -3.0000, A 0.000, B 0.000, C 0.000 }
gfCNCPoint2[23276] = {X 559.0942, Y 8.5330, Z -3.0000, A 0.000, B 0.000, C 0.000 }
gfCNCPoint2[23277] = {X 558.6132, Y 7.7507, Z -3.0000, A 0.000, B 0.000, C 0.000 }
gfCNCPoint2[23278] = {X 558.3119, Y 6.8832, Z -3.0000, A 0.000, B 0.000, C 0.000 }
gfCNCPoint2[23279] = {X 558.2045, Y 5.9711, Z -3.0000, A 0.000, B 0.000, C 0.000 }
gfCNCPoint2[23280] = {X 558.2043, Y 5.0000, Z -3.0000, A 0.000, B 0.000, C 0.000 }
gfCNCPoint2[23281] = {X 558.3106, Y 4.0565, Z -3.0000, A 0.000, B 0.000, C 0.000 }
gfCNCPoint2[23282] = {X 558.6242, Y 3.1603, Z -3.0000, A 0.000, B 0.000, C 0.000 }
gfCNCPoint2[23283] = {X 559.1293, Y 2.3564, Z -3.0000, A 0.000, B 0.000, C 0.000 }
gfCNCPoint2[23284] = {X 559.8007, Y 1.6850, Z -3.0000, A 0.000, B 0.000, C 0.000 }
gfCNCPoint2[23285] = {X 560.6046, Y 1.1799, Z -3.0000, A 0.000, B 0.000, C 0.000 }
gfCNCPoint2[23286] = {X 561.5008, Y 0.8663, Z -3.0000, A 0.000, B 0.000, C 0.000 }
gfCNCPoint2[23287] = {X 562.4443, Y 0.7600, Z -3.0000, A 0.000, B 0.000, C 0.000 }
gfCNCPoint2[23288] = {X 570.9376, Y 0.7600, Z -3.0000, A 0.000, B 0.000, C 0.000 }
gfCNCPoint2[23289] = {X 571.8810, Y 0.8663, Z -3.0000, A 0.000, B 0.000, C 0.000 }
gfCNCPoint2[23290] = {X 572.7772, Y 1.1799, Z -3.0000, A 0.000, B 0.000, C 0.000 }
gfCNCPoint2[23291] = {X 573.5812, Y 1.6850, Z -3.0000, A 0.000, B 0.000, C 0.000 }
gfCNCPoint2[23292] = {X 574.2525, Y 2.3564, Z -3.0000, A 0.000, B 0.000, C 0.000 }
gfCNCPoint2[23293] = {X 574.7577, Y 3.1603, Z -3.0000, A 0.000, B 0.000, C 0.000 }
gfCNCPoint2[23294] = {X 575.0712, Y 4.0565, Z -3.0000, A 0.000, B 0.000, C 0.000 }
gfCNCPoint2[23295] = {X 575.1776, Y 5.0000, Z -3.0000, A 0.000, B 0.000, C 0.000 }
gfCNCPoint2[23296] = {X 575.1776, Y 5.9342, Z -3.0000, A 0.000, B 0.000, C 0.000 }
gfCNCPoint2[23297] = {X 575.1023, Y 6.7293, Z -3.0000, A 0.000, B 0.000, C 0.000 }
gfCNCPoint2[23298] = {X 574.8793, Y 7.4961, Z -3.0000, A 0.000, B 0.000, C 0.000 }
gfCNCPoint2[23299] = {X 574.5165, Y 8.2075, Z -3.0000, A 0.000, B 0.000, C 0.000 }
gfCNCPoint2[23300] = {X 581.1908, Y 24.5822, Z -3.0000, A 0.000, B 0.000, C 0.000 }
gfCNCPoint2[23301] = {X 587.9349, Y 8.0882, Z -3.0000, A 0.000, B 0.000, C 0.000 }
gfCNCPoint2[23302] = {X 587.6159, Y 7.4201, Z -3.0000, A 0.000, B 0.000, C 0.000 }
gfCNCPoint2[23303] = {X 587.4180, Y 6.7067, Z -3.0000, A 0.000, B 0.000, C 0.000 }
gfCNCPoint2[23304] = {X 587.3471, Y 5.9698, Z -3.0000, A 0.000, B 0.000, C 0.000 }
gfCNCPoint2[23305] = {X 587.3470, Y 5.0000, Z -3.0000, A 0.000, B 0.000, C 0.000 }
gfCNCPoint2[23306] = {X 587.4533, Y 4.0565, Z -3.0000, A 0.000, B 0.000, C 0.000 }
gfCNCPoint2[23307] = {X 587.7668, Y 3.1603, Z -3.0000, A 0.000, B 0.000, C 0.000 }
gfCNCPoint2[23308] = {X 588.2720, Y 2.3564, Z -3.0000, A 0.000, B 0.000, C 0.000 }
gfCNCPoint2[23309] = {X 588.9434, Y 1.6850, Z -3.0000, A 0.000, B 0.000, C 0.000 }
gfCNCPoint2[23310] = {X 589.7473, Y 1.1799, Z -3.0000, A 0.000, B 0.000, C 0.000 }
gfCNCPoint2[23311] = {X 590.6435, Y 0.8663, Z -3.0000, A 0.000, B 0.000, C 0.000 }
gfCNCPoint2[23312] = {X 591.5870, Y 0.7600, Z -3.0000, A 0.000, B 0.000, C 0.000 }
gfCNCPoint2[23313] = {X 600.0000, Y 0.7600, Z -3.0000, A 0.000, B 0.000, C 0.000 }
gfCNCPoint2[23314] = {X 600.8403, Y 0.8441, Z -3.0000, A 0.000, B 0.000, C 0.000 }
gfCNCPoint2[23315] = {X 601.6472, Y 1.0931, Z -3.0000, A 0.000, B 0.000, C 0.000 }
gfCNCPoint2[23316] = {X 602.3888, Y 1.4970, Z -3.0000, A 0.000, B 0.000, C 0.000 }
gfCNCPoint2[23317] = {X 603.0357, Y 2.0399, Z -3.0000, A 0.000, B 0.000, C 0.000 }
gfCNCPoint2[23318] = {X 603.5621, Y 2.7002, Z -3.0000, A 0.000, B 0.000, C 0.000 }
gfCNCPoint2[23319] = {X 603.6310, Y 2.8106, Z -3.0000, A 0.000, B 0.000, C 0.000 }
gfCNCPoint2[23320] = {X 603.6965, Y 2.9231, Z -3.0000, A 0.000, B 0.000, C 0.000 }
gfCNCPoint2[23321] = {X 607.8232, Y 10.2681, Z -3.0000, A 0.000, B 0.000, C 0.000 }
gfCNCPoint2[23322] = {X 607.8232, Y 10.2681, Z 0.0000, A 0.000, B 0.000, C 0.000 }
gfCNCPoint2[23323] = {X 607.8232, Y 10.2681, Z 11.0000, A 0.000, B 0.000, C 0.000 }
gfCNCPoint2[23324] = {X 607.6965, Y 39.1597, Z 11.0000, A 0.000, B 0.000, C 0.000 }
gfCNCPoint2[23325] = {X 607.6965, Y 39.1597, Z 0.0000, A 0.000, B 0.000, C 0.000 }
gfCNCPoint2[23326] = {X 607.6965, Y 39.1597, Z -3.0000, A 0.000, B 0.000, C 0.000 }
gfCNCPoint2[23327] = {X 603.6965, Y 46.9082, Z -3.0000, A 0.000, B 0.000, C 0.000 }
gfCNCPoint2[23328] = {X 603.5999, Y 47.0848, Z -3.0000, A 0.000, B 0.000, C 0.000 }
gfCNCPoint2[23329] = {X 603.4949, Y 47.2564, Z -3.0000, A 0.000, B 0.000, C 0.000 }
gfCNCPoint2[23330] = {X 602.9784, Y 47.9043, Z -3.0000, A 0.000, B 0.000, C 0.000 }
gfCNCPoint2[23331] = {X 602.3438, Y 48.4369, Z -3.0000, A 0.000, B 0.000, C 0.000 }
gfCNCPoint2[23332] = {X 601.6161, Y 48.8332, Z -3.0000, A 0.000, B 0.000, C 0.000 }
gfCNCPoint2[23333] = {X 600.8244, Y 49.0775, Z -3.0000, A 0.000, B 0.000, C 0.000 }
gfCNCPoint2[23334] = {X 600.0000, Y 49.1600, Z -3.0000, A 0.000, B 0.000, C 0.000 }
gfCNCPoint2[23335] = {X 593.5565, Y 49.1600, Z -3.0000, A 0.000, B 0.000, C 0.000 }
gfCNCPoint2[23336] = {X 592.6308, Y 49.0557, Z -3.0000, A 0.000, B 0.000, C 0.000 }
gfCNCPoint2[23337] = {X 591.7516, Y 48.7480, Z -3.0000, A 0.000, B 0.000, C 0.000 }
gfCNCPoint2[23338] = {X 590.9628, Y 48.2524, Z -3.0000, A 0.000, B 0.000, C 0.000 }
gfCNCPoint2[23339] = {X 590.3041, Y 47.5937, Z -3.0000, A 0.000, B 0.000, C 0.000 }
gfCNCPoint2[23340] = {X 589.8085, Y 46.8050, Z -3.0000, A 0.000, B 0.000, C 0.000 }
gfCNCPoint2[23341] = {X 589.5008, Y 45.9257, Z -3.0000, A 0.000, B 0.000, C 0.000 }
gfCNCPoint2[23342] = {X 589.3965, Y 45.0000, Z -3.0000, A 0.000, B 0.000, C 0.000 }
gfCNCPoint2[23343] = {X 589.3965, Y 44.0652, Z -3.0000, A 0.000, B 0.000, C 0.000 }
gfCNCPoint2[23344] = {X 589.5014, Y 43.1533, Z -3.0000, A 0.000, B 0.000, C 0.000 }
gfCNCPoint2[23345] = {X 589.8017, Y 42.2859, Z -3.0000, A 0.000, B 0.000, C 0.000 }
gfCNCPoint2[23346] = {X 590.2831, Y 41.5044, Z -3.0000, A 0.000, B 0.000, C 0.000 }
gfCNCPoint2[23347] = {X 590.9228, Y 40.8460, Z -3.0000, A 0.000, B 0.000, C 0.000 }
gfCNCPoint2[23348] = {X 590.9232, Y 32.7089, Z -3.0000, A 0.000, B 0.000, C 0.000 }
gfCNCPoint2[23349] = {X 585.2975, Y 46.5912, Z -3.0000, A 0.000, B 0.000, C 0.000 }
gfCNCPoint2[23350] = {X 584.9414, Y 47.2678, Z -3.0000, A 0.000, B 0.000, C 0.000 }
gfCNCPoint2[23351] = {X 584.4675, Y 47.8677, Z -3.0000, A 0.000, B 0.000, C 0.000 }
gfCNCPoint2[23352] = {X 583.8918, Y 48.3708, Z -3.0000, A 0.000, B 0.000, C 0.000 }
gfCNCPoint2[23353] = {X 583.2338, Y 48.7600, Z -3.0000, A 0.000, B 0.000, C 0.000 }
gfCNCPoint2[23354] = {X 582.3250, Y 49.0678, Z -3.0000, A 0.000, B 0.000, C 0.000 }
gfCNCPoint2[23355] = {X 581.3699, Y 49.1592, Z -3.0000, A 0.000, B 0.000, C 0.000 }
gfCNCPoint2[23356] = {X 580.4192, Y 49.0293, Z -3.0000, A 0.000, B 0.000, C 0.000 }
gfCNCPoint2[23357] = {X 579.5236, Y 48.6850, Z -3.0000, A 0.000, B 0.000, C 0.000 }
gfCNCPoint2[23358] = {X 578.7306, Y 48.1448, Z -3.0000, A 0.000, B 0.000, C 0.000 }
gfCNCPoint2[23359] = {X 578.0826, Y 47.4372, Z -3.0000, A 0.000, B 0.000, C 0.000 }
gfCNCPoint2[23360] = {X 577.6138, Y 46.5999, Z -3.0000, A 0.000, B 0.000, C 0.000 }
gfCNCPoint2[23361] = {X 571.8582, Y 32.5259, Z -3.0000, A 0.000, B 0.000, C 0.000 }
gfCNCPoint2[23362] = {X 571.8586, Y 40.8460, Z -3.0000, A 0.000, B 0.000, C 0.000 }
gfCNCPoint2[23363] = {X 571.9194, Y 40.8952, Z -3.0000, A 0.000, B 0.000, C 0.000 }
gfCNCPoint2[23364] = {X 572.5327, Y 41.5412, Z -3.0000, A 0.000, B 0.000, C 0.000 }
gfCNCPoint2[23365] = {X 572.9943, Y 42.3029, Z -3.0000, A 0.000, B 0.000, C 0.000 }
gfCNCPoint2[23366] = {X 573.2833, Y 43.1454, Z -3.0000, A 0.000, B 0.000, C 0.000 }
gfCNCPoint2[23367] = {X 573.3863, Y 44.0301, Z -3.0000, A 0.000, B 0.000, C 0.000 }
gfCNCPoint2[23368] = {X 573.3864, Y 45.0000, Z -3.0000, A 0.000, B 0.000, C 0.000 }
gfCNCPoint2[23369] = {X 573.2821, Y 45.9257, Z -3.0000, A 0.000, B 0.000, C 0.000 }
gfCNCPoint2[23370] = {X 572.9745, Y 46.8050, Z -3.0000, A 0.000, B 0.000, C 0.000 }
gfCNCPoint2[23371] = {X 572.4788, Y 47.5937, Z -3.0000, A 0.000, B 0.000, C 0.000 }
gfCNCPoint2[23372] = {X 571.8201, Y 48.2524, Z -3.0000, A 0.000, B 0.000, C 0.000 }
gfCNCPoint2[23373] = {X 571.0314, Y 48.7480, Z -3.0000, A 0.000, B 0.000, C 0.000 }
gfCNCPoint2[23374] = {X 570.1521, Y 49.0557, Z -3.0000, A 0.000, B 0.000, C 0.000 }
gfCNCPoint2[23375] = {X 569.2264, Y 49.1600, Z -3.0000, A 0.000, B 0.000, C 0.000 }
gfCNCPoint2[23376] = {X 562.4443, Y 49.1600, Z -3.0000, A 0.000, B 0.000, C 0.000 }
gfCNCPoint2[23377] = {X 561.5186, Y 49.0557, Z -3.0000, A 0.000, B 0.000, C 0.000 }
gfCNCPoint2[23378] = {X 560.6393, Y 48.7480, Z -3.0000, A 0.000, B 0.000, C 0.000 }
gfCNCPoint2[23379] = {X 559.8506, Y 48.2524, Z -3.0000, A 0.000, B 0.000, C 0.000 }
gfCNCPoint2[23380] = {X 559.1919, Y 47.5937, Z -3.0000, A 0.000, B 0.000, C 0.000 }
gfCNCPoint2[23381] = {X 558.6963, Y 46.8050, Z -3.0000, A 0.000, B 0.000, C 0.000 }
gfCNCPoint2[23382] = {X 558.3886, Y 45.9257, Z -3.0000, A 0.000, B 0.000, C 0.000 }
gfCNCPoint2[23383] = {X 558.2843, Y 45.0000, Z -3.0000, A 0.000, B 0.000, C 0.000 }
gfCNCPoint2[23384] = {X 558.2843, Y 44.0653, Z -3.0000, A 0.000, B 0.000, C 0.000 }
gfCNCPoint2[23385] = {X 558.3890, Y 43.1530, Z -3.0000, A 0.000, B 0.000, C 0.000 }
gfCNCPoint2[23386] = {X 558.6896, Y 42.2853, Z -3.0000, A 0.000, B 0.000, C 0.000 }
gfCNCPoint2[23387] = {X 559.1718, Y 41.5037, Z -3.0000, A 0.000, B 0.000, C 0.000 }
gfCNCPoint2[23388] = {X 559.8124, Y 40.8458, Z -3.0000, A 0.000, B 0.000, C 0.000 }
gfCNCPoint2[23389] = {X 559.8124, Y 9.1556, Z -3.0000, A 0.000, B 0.000, C 0.000 }
gfCNCPoint2[23390] = {X 559.1747, Y 8.5060, Z -3.0000, A 0.000, B 0.000, C 0.000 }
gfCNCPoint2[23391] = {X 558.6935, Y 7.7333, Z -3.0000, A 0.000, B 0.000, C 0.000 }
gfCNCPoint2[23392] = {X 558.3920, Y 6.8744, Z -3.0000, A 0.000, B 0.000, C 0.000 }
gfCNCPoint2[23393] = {X 558.2845, Y 5.9704, Z -3.0000, A 0.000, B 0.000, C 0.000 }
gfCNCPoint2[23394] = {X 558.2843, Y 5.0000, Z -3.0000, A 0.000, B 0.000, C 0.000 }
gfCNCPoint2[23395] = {X 558.3886, Y 4.0743, Z -3.0000, A 0.000, B 0.000, C 0.000 }
gfCNCPoint2[23396] = {X 558.6963, Y 3.1950, Z -3.0000, A 0.000, B 0.000, C 0.000 }
gfCNCPoint2[23397] = {X 559.1919, Y 2.4063, Z -3.0000, A 0.000, B 0.000, C 0.000 }
gfCNCPoint2[23398] = {X 559.8506, Y 1.7476, Z -3.0000, A 0.000, B 0.000, C 0.000 }
gfCNCPoint2[23399] = {X 560.6393, Y 1.2520, Z -3.0000, A 0.000, B 0.000, C 0.000 }
gfCNCPoint2[23400] = {X 561.5186, Y 0.9443, Z -3.0000, A 0.000, B 0.000, C 0.000 }
gfCNCPoint2[23401] = {X 562.4443, Y 0.8400, Z -3.0000, A 0.000, B 0.000, C 0.000 }
gfCNCPoint2[23402] = {X 570.9376, Y 0.8400, Z -3.0000, A 0.000, B 0.000, C 0.000 }
gfCNCPoint2[23403] = {X 571.8632, Y 0.9443, Z -3.0000, A 0.000, B 0.000, C 0.000 }
gfCNCPoint2[23404] = {X 572.7425, Y 1.2520, Z -3.0000, A 0.000, B 0.000, C 0.000 }
gfCNCPoint2[23405] = {X 573.5313, Y 1.7476, Z -3.0000, A 0.000, B 0.000, C 0.000 }
gfCNCPoint2[23406] = {X 574.1900, Y 2.4063, Z -3.0000, A 0.000, B 0.000, C 0.000 }
gfCNCPoint2[23407] = {X 574.6856, Y 3.1950, Z -3.0000, A 0.000, B 0.000, C 0.000 }
gfCNCPoint2[23408] = {X 574.9933, Y 4.0743, Z -3.0000, A 0.000, B 0.000, C 0.000 }
gfCNCPoint2[23409] = {X 575.0976, Y 5.0000, Z -3.0000, A 0.000, B 0.000, C 0.000 }
gfCNCPoint2[23410] = {X 575.0976, Y 5.9342, Z -3.0000, A 0.000, B 0.000, C 0.000 }
gfCNCPoint2[23411] = {X 575.0211, Y 6.7277, Z -3.0000, A 0.000, B 0.000, C 0.000 }
gfCNCPoint2[23412] = {X 574.7948, Y 7.4921, Z -3.0000, A 0.000, B 0.000, C 0.000 }
gfCNCPoint2[23413] = {X 574.4268, Y 8.1992, Z -3.0000, A 0.000, B 0.000, C 0.000 }
gfCNCPoint2[23414] = {X 581.1907, Y 24.7939, Z -3.0000, A 0.000, B 0.000, C 0.000 }
gfCNCPoint2[23415] = {X 588.0241, Y 8.0815, Z -3.0000, A 0.000, B 0.000, C 0.000 }
gfCNCPoint2[23416] = {X 587.7001, Y 7.4167, Z -3.0000, A 0.000, B 0.000, C 0.000 }
gfCNCPoint2[23417] = {X 587.4990, Y 6.7051, Z -3.0000, A 0.000, B 0.000, C 0.000 }
gfCNCPoint2[23418] = {X 587.4271, Y 5.9692, Z -3.0000, A 0.000, B 0.000, C 0.000 }
gfCNCPoint2[23419] = {X 587.4270, Y 5.0000, Z -3.0000, A 0.000, B 0.000, C 0.000 }
gfCNCPoint2[23420] = {X 587.5313, Y 4.0743, Z -3.0000, A 0.000, B 0.000, C 0.000 }
gfCNCPoint2[23421] = {X 587.8389, Y 3.1950, Z -3.0000, A 0.000, B 0.000, C 0.000 }
gfCNCPoint2[23422] = {X 588.3345, Y 2.4063, Z -3.0000, A 0.000, B 0.000, C 0.000 }
gfCNCPoint2[23423] = {X 588.9932, Y 1.7476, Z -3.0000, A 0.000, B 0.000, C 0.000 }
gfCNCPoint2[23424] = {X 589.7820, Y 1.2520, Z -3.0000, A 0.000, B 0.000, C 0.000 }
gfCNCPoint2[23425] = {X 590.6613, Y 0.9443, Z -3.0000, A 0.000, B 0.000, C 0.000 }
gfCNCPoint2[23426] = {X 591.5870, Y 0.8400, Z -3.0000, A 0.000, B 0.000, C 0.000 }
gfCNCPoint2[23427] = {X 600.0000, Y 0.8400, Z -3.0000, A 0.000, B 0.000, C 0.000 }
gfCNCPoint2[23428] = {X 600.8244, Y 0.9225, Z -3.0000, A 0.000, B 0.000, C 0.000 }
gfCNCPoint2[23429] = {X 601.6161, Y 1.1668, Z -3.0000, A 0.000, B 0.000, C 0.000 }
gfCNCPoint2[23430] = {X 602.3438, Y 1.5631, Z -3.0000, A 0.000, B 0.000, C 0.000 }
gfCNCPoint2[23431] = {X 602.9784, Y 2.0957, Z -3.0000, A 0.000, B 0.000, C 0.000 }
gfCNCPoint2[23432] = {X 603.4949, Y 2.7436, Z -3.0000, A 0.000, B 0.000, C 0.000 }
gfCNCPoint2[23433] = {X 603.5999, Y 2.9152, Z -3.0000, A 0.000, B 0.000, C 0.000 }
gfCNCPoint2[23434] = {X 603.6965, Y 3.0918, Z -3.0000, A 0.000, B 0.000, C 0.000 }
gfCNCPoint2[23435] = {X 607.6965, Y 10.8403, Z -3.0000, A 0.000, B 0.000, C 0.000 }
gfCNCPoint2[23436] = {X 607.6965, Y 10.8403, Z 0.0000, A 0.000, B 0.000, C 0.000 }
gfCNCPoint2[23437] = {X 607.6965, Y 10.8403, Z 11.0000, A 0.000, B 0.000, C 0.000 }
gfCNCPoint2[23438] = {X 607.6965, Y 38.1647, Z 11.0000, A 0.000, B 0.000, C 0.000 }
gfCNCPoint2[23439] = {X 607.6965, Y 38.1647, Z 0.0000, A 0.000, B 0.000, C 0.000 }
gfCNCPoint2[23440] = {X 607.6965, Y 38.1647, Z -3.0000, A 0.000, B 0.000, C 0.000 }
gfCNCPoint2[23441] = {X 603.6965, Y 46.7269, Z -3.0000, A 0.000, B 0.000, C 0.000 }
gfCNCPoint2[23442] = {X 603.5704, Y 46.9745, Z -3.0000, A 0.000, B 0.000, C 0.000 }
gfCNCPoint2[23443] = {X 603.4277, Y 47.2130, Z -3.0000, A 0.000, B 0.000, C 0.000 }
gfCNCPoint2[23444] = {X 602.9211, Y 47.8484, Z -3.0000, A 0.000, B 0.000, C 0.000 }
gfCNCPoint2[23445] = {X 602.2987, Y 48.3708, Z -3.0000, A 0.000, B 0.000, C 0.000 }
gfCNCPoint2[23446] = {X 601.5851, Y 48.7595, Z -3.0000, A 0.000, B 0.000, C 0.000 }
gfCNCPoint2[23447] = {X 600.8086, Y 48.9991, Z -3.0000, A 0.000, B 0.000, C 0.000 }
gfCNCPoint2[23448] = {X 600.0000, Y 49.0800, Z -3.0000, A 0.000, B 0.000, C 0.000 }
gfCNCPoint2[23449] = {X 593.5565, Y 49.0800, Z -3.0000, A 0.000, B 0.000, C 0.000 }
gfCNCPoint2[23450] = {X 592.6486, Y 48.9777, Z -3.0000, A 0.000, B 0.000, C 0.000 }
gfCNCPoint2[23451] = {X 591.7863, Y 48.6760, Z -3.0000, A 0.000, B 0.000, C 0.000 }
gfCNCPoint2[23452] = {X 591.0127, Y 48.1899, Z -3.0000, A 0.000, B 0.000, C 0.000 }
gfCNCPoint2[23453] = {X 590.3667, Y 47.5438, Z -3.0000, A 0.000, B 0.000, C 0.000 }
gfCNCPoint2[23454] = {X 589.8806, Y 46.7702, Z -3.0000, A 0.000, B 0.000, C 0.000 }
gfCNCPoint2[23455] = {X 589.5788, Y 45.9079, Z -3.0000, A 0.000, B 0.000, C 0.000 }
gfCNCPoint2[23456] = {X 589.4765, Y 45.0000, Z -3.0000, A 0.000, B 0.000, C 0.000 }
gfCNCPoint2[23457] = {X 589.4765, Y 44.0656, Z -3.0000, A 0.000, B 0.000, C 0.000 }
gfCNCPoint2[23458] = {X 589.5815, Y 43.1619, Z -3.0000, A 0.000, B 0.000, C 0.000 }
gfCNCPoint2[23459] = {X 589.8821, Y 42.3032, Z -3.0000, A 0.000, B 0.000, C 0.000 }
gfCNCPoint2[23460] = {X 590.3636, Y 41.5314, Z -3.0000, A 0.000, B 0.000, C 0.000 }
gfCNCPoint2[23461] = {X 591.0028, Y 40.8839, Z -3.0000, A 0.000, B 0.000, C 0.000 }
gfCNCPoint2[23462] = {X 591.0033, Y 32.2985, Z -3.0000, A 0.000, B 0.000, C 0.000 }
gfCNCPoint2[23463] = {X 585.2236, Y 46.5606, Z -3.0000, A 0.000, B 0.000, C 0.000 }
gfCNCPoint2[23464] = {X 584.8743, Y 47.2242, Z -3.0000, A 0.000, B 0.000, C 0.000 }
gfCNCPoint2[23465] = {X 584.4095, Y 47.8125, Z -3.0000, A 0.000, B 0.000, C 0.000 }
gfCNCPoint2[23466] = {X 583.8449, Y 48.3059, Z -3.0000, A 0.000, B 0.000, C 0.000 }
gfCNCPoint2[23467] = {X 583.1996, Y 48.6877, Z -3.0000, A 0.000, B 0.000, C 0.000 }
gfCNCPoint2[23468] = {X 582.3082, Y 48.9895, Z -3.0000, A 0.000, B 0.000, C 0.000 }
gfCNCPoint2[23469] = {X 581.3715, Y 49.0792, Z -3.0000, A 0.000, B 0.000, C 0.000 }
gfCNCPoint2[23470] = {X 580.4391, Y 48.9518, Z -3.0000, A 0.000, B 0.000, C 0.000 }
gfCNCPoint2[23471] = {X 579.5607, Y 48.6142, Z -3.0000, A 0.000, B 0.000, C 0.000 }
gfCNCPoint2[23472] = {X 578.7830, Y 48.0843, Z -3.0000, A 0.000, B 0.000, C 0.000 }
gfCNCPoint2[23473] = {X 578.1474, Y 47.3903, Z -3.0000, A 0.000, B 0.000, C 0.000 }
gfCNCPoint2[23474] = {X 577.6877, Y 46.5692, Z -3.0000, A 0.000, B 0.000, C 0.000 }
gfCNCPoint2[23475] = {X 571.7782, Y 32.1189, Z -3.0000, A 0.000, B 0.000, C 0.000 }
gfCNCPoint2[23476] = {X 571.7786, Y 40.8842, Z -3.0000, A 0.000, B 0.000, C 0.000 }
gfCNCPoint2[23477] = {X 571.8683, Y 40.9568, Z -3.0000, A 0.000, B 0.000, C 0.000 }
gfCNCPoint2[23478] = {X 572.4695, Y 41.5903, Z -3.0000, A 0.000, B 0.000, C 0.000 }
gfCNCPoint2[23479] = {X 572.9221, Y 42.3372, Z -3.0000, A 0.000, B 0.000, C 0.000 }
gfCNCPoint2[23480] = {X 573.2053, Y 43.1633, Z -3.0000, A 0.000, B 0.000, C 0.000 }
gfCNCPoint2[23481] = {X 573.3063, Y 44.0308, Z -3.0000, A 0.000, B 0.000, C 0.000 }
gfCNCPoint2[23482] = {X 573.3064, Y 45.0000, Z -3.0000, A 0.000, B 0.000, C 0.000 }
gfCNCPoint2[23483] = {X 573.2041, Y 45.9079, Z -3.0000, A 0.000, B 0.000, C 0.000 }
gfCNCPoint2[23484] = {X 572.9024, Y 46.7702, Z -3.0000, A 0.000, B 0.000, C 0.000 }
gfCNCPoint2[23485] = {X 572.4163, Y 47.5438, Z -3.0000, A 0.000, B 0.000, C 0.000 }
gfCNCPoint2[23486] = {X 571.7703, Y 48.1899, Z -3.0000, A 0.000, B 0.000, C 0.000 }
gfCNCPoint2[23487] = {X 570.9967, Y 48.6760, Z -3.0000, A 0.000, B 0.000, C 0.000 }
gfCNCPoint2[23488] = {X 570.1343, Y 48.9777, Z -3.0000, A 0.000, B 0.000, C 0.000 }
gfCNCPoint2[23489] = {X 569.2264, Y 49.0800, Z -3.0000, A 0.000, B 0.000, C 0.000 }
gfCNCPoint2[23490] = {X 562.4443, Y 49.0800, Z -3.0000, A 0.000, B 0.000, C 0.000 }
gfCNCPoint2[23491] = {X 561.5364, Y 48.9777, Z -3.0000, A 0.000, B 0.000, C 0.000 }
gfCNCPoint2[23492] = {X 560.6741, Y 48.6760, Z -3.0000, A 0.000, B 0.000, C 0.000 }
gfCNCPoint2[23493] = {X 559.9005, Y 48.1899, Z -3.0000, A 0.000, B 0.000, C 0.000 }
gfCNCPoint2[23494] = {X 559.2544, Y 47.5438, Z -3.0000, A 0.000, B 0.000, C 0.000 }
gfCNCPoint2[23495] = {X 558.7683, Y 46.7702, Z -3.0000, A 0.000, B 0.000, C 0.000 }
gfCNCPoint2[23496] = {X 558.4666, Y 45.9079, Z -3.0000, A 0.000, B 0.000, C 0.000 }
gfCNCPoint2[23497] = {X 558.3643, Y 45.0000, Z -3.0000, A 0.000, B 0.000, C 0.000 }
gfCNCPoint2[23498] = {X 558.3643, Y 44.0656, Z -3.0000, A 0.000, B 0.000, C 0.000 }
gfCNCPoint2[23499] = {X 558.4612, Y 43.1966, Z -3.0000, A 0.000, B 0.000, C 0.000 }
gfCNCPoint2[23500] = {X 558.7394, Y 42.3677, Z -3.0000, A 0.000, B 0.000, C 0.000 }
gfCNCPoint2[23501] = {X 559.1865, Y 41.6162, Z -3.0000, A 0.000, B 0.000, C 0.000 }
gfCNCPoint2[23502] = {X 559.7822, Y 40.9761, Z -3.0000, A 0.000, B 0.000, C 0.000 }
gfCNCPoint2[23503] = {X 559.8369, Y 40.9295, Z -3.0000, A 0.000, B 0.000, C 0.000 }
gfCNCPoint2[23504] = {X 559.8924, Y 40.8838, Z -3.0000, A 0.000, B 0.000, C 0.000 }
gfCNCPoint2[23505] = {X 559.8924, Y 9.1175, Z -3.0000, A 0.000, B 0.000, C 0.000 }
gfCNCPoint2[23506] = {X 559.2551, Y 8.4788, Z -3.0000, A 0.000, B 0.000, C 0.000 }
gfCNCPoint2[23507] = {X 558.7739, Y 7.7157, Z -3.0000, A 0.000, B 0.000, C 0.000 }
gfCNCPoint2[23508] = {X 558.4720, Y 6.8655, Z -3.0000, A 0.000, B 0.000, C 0.000 }
gfCNCPoint2[23509] = {X 558.3645, Y 5.9697, Z -3.0000, A 0.000, B 0.000, C 0.000 }
gfCNCPoint2[23510] = {X 558.3643, Y 5.0000, Z -3.0000, A 0.000, B 0.000, C 0.000 }
gfCNCPoint2[23511] = {X 558.4666, Y 4.0921, Z -3.0000, A 0.000, B 0.000, C 0.000 }
gfCNCPoint2[23512] = {X 558.7683, Y 3.2298, Z -3.0000, A 0.000, B 0.000, C 0.000 }
gfCNCPoint2[23513] = {X 559.2544, Y 2.4562, Z -3.0000, A 0.000, B 0.000, C 0.000 }
gfCNCPoint2[23514] = {X 559.9005, Y 1.8101, Z -3.0000, A 0.000, B 0.000, C 0.000 }
gfCNCPoint2[23515] = {X 560.6741, Y 1.3240, Z -3.0000, A 0.000, B 0.000, C 0.000 }
gfCNCPoint2[23516] = {X 561.5364, Y 1.0223, Z -3.0000, A 0.000, B 0.000, C 0.000 }
gfCNCPoint2[23517] = {X 562.4443, Y 0.9200, Z -3.0000, A 0.000, B 0.000, C 0.000 }
gfCNCPoint2[23518] = {X 570.9376, Y 0.9200, Z -3.0000, A 0.000, B 0.000, C 0.000 }
gfCNCPoint2[23519] = {X 571.8454, Y 1.0223, Z -3.0000, A 0.000, B 0.000, C 0.000 }
gfCNCPoint2[23520] = {X 572.7078, Y 1.3240, Z -3.0000, A 0.000, B 0.000, C 0.000 }
gfCNCPoint2[23521] = {X 573.4814, Y 1.8101, Z -3.0000, A 0.000, B 0.000, C 0.000 }
gfCNCPoint2[23522] = {X 574.1274, Y 2.4562, Z -3.0000, A 0.000, B 0.000, C 0.000 }
gfCNCPoint2[23523] = {X 574.6135, Y 3.2298, Z -3.0000, A 0.000, B 0.000, C 0.000 }
gfCNCPoint2[23524] = {X 574.9153, Y 4.0921, Z -3.0000, A 0.000, B 0.000, C 0.000 }
gfCNCPoint2[23525] = {X 575.0176, Y 5.0000, Z -3.0000, A 0.000, B 0.000, C 0.000 }
gfCNCPoint2[23526] = {X 575.0176, Y 5.9342, Z -3.0000, A 0.000, B 0.000, C 0.000 }
gfCNCPoint2[23527] = {X 574.9499, Y 6.6738, Z -3.0000, A 0.000, B 0.000, C 0.000 }
gfCNCPoint2[23528] = {X 574.7494, Y 7.3888, Z -3.0000, A 0.000, B 0.000, C 0.000 }
gfCNCPoint2[23529] = {X 574.4226, Y 8.0557, Z -3.0000, A 0.000, B 0.000, C 0.000 }
gfCNCPoint2[23530] = {X 574.3782, Y 8.1268, Z -3.0000, A 0.000, B 0.000, C 0.000 }
gfCNCPoint2[23531] = {X 574.3324, Y 8.1971, Z -3.0000, A 0.000, B 0.000, C 0.000 }
gfCNCPoint2[23532] = {X 574.3582, Y 8.2420, Z -3.0000, A 0.000, B 0.000, C 0.000 }
gfCNCPoint2[23533] = {X 581.1906, Y 25.0055, Z -3.0000, A 0.000, B 0.000, C 0.000 }
gfCNCPoint2[23534] = {X 588.1134, Y 8.0744, Z -3.0000, A 0.000, B 0.000, C 0.000 }
gfCNCPoint2[23535] = {X 587.7845, Y 7.4131, Z -3.0000, A 0.000, B 0.000, C 0.000 }
gfCNCPoint2[23536] = {X 587.5801, Y 6.7034, Z -3.0000, A 0.000, B 0.000, C 0.000 }
gfCNCPoint2[23537] = {X 587.5071, Y 5.9685, Z -3.0000, A 0.000, B 0.000, C 0.000 }
gfCNCPoint2[23538] = {X 587.5070, Y 5.0000, Z -3.0000, A 0.000, B 0.000, C 0.000 }
gfCNCPoint2[23539] = {X 587.6092, Y 4.0921, Z -3.0000, A 0.000, B 0.000, C 0.000 }
gfCNCPoint2[23540] = {X 587.9110, Y 3.2298, Z -3.0000, A 0.000, B 0.000, C 0.000 }
gfCNCPoint2[23541] = {X 588.3971, Y 2.4562, Z -3.0000, A 0.000, B 0.000, C 0.000 }
gfCNCPoint2[23542] = {X 589.0431, Y 1.8101, Z -3.0000, A 0.000, B 0.000, C 0.000 }
gfCNCPoint2[23543] = {X 589.8167, Y 1.3240, Z -3.0000, A 0.000, B 0.000, C 0.000 }
gfCNCPoint2[23544] = {X 590.6791, Y 1.0223, Z -3.0000, A 0.000, B 0.000, C 0.000 }
gfCNCPoint2[23545] = {X 591.5870, Y 0.9200, Z -3.0000, A 0.000, B 0.000, C 0.000 }
gfCNCPoint2[23546] = {X 600.0000, Y 0.9200, Z -3.0000, A 0.000, B 0.000, C 0.000 }
gfCNCPoint2[23547] = {X 600.8086, Y 1.0009, Z -3.0000, A 0.000, B 0.000, C 0.000 }
gfCNCPoint2[23548] = {X 601.5851, Y 1.2405, Z -3.0000, A 0.000, B 0.000, C 0.000 }
gfCNCPoint2[23549] = {X 602.2987, Y 1.6292, Z -3.0000, A 0.000, B 0.000, C 0.000 }
gfCNCPoint2[23550] = {X 602.9211, Y 2.1516, Z -3.0000, A 0.000, B 0.000, C 0.000 }
gfCNCPoint2[23551] = {X 603.4277, Y 2.7870, Z -3.0000, A 0.000, B 0.000, C 0.000 }
gfCNCPoint2[23552] = {X 603.5704, Y 3.0255, Z -3.0000, A 0.000, B 0.000, C 0.000 }
gfCNCPoint2[23553] = {X 603.6965, Y 3.2731, Z -3.0000, A 0.000, B 0.000, C 0.000 }
gfCNCPoint2[23554] = {X 607.6965, Y 11.8353, Z -3.0000, A 0.000, B 0.000, C 0.000 }
gfCNCPoint2[23555] = {X 607.6965, Y 11.8353, Z 0.0000, A 0.000, B 0.000, C 0.000 }
gfCNCPoint2[23556] = {X 607.6965, Y 11.8353, Z 11.0000, A 0.000, B 0.000, C 0.000 }
gfCNCPoint2[23557] = {X 607.6965, Y 36.8536, Z 11.0000, A 0.000, B 0.000, C 0.000 }
gfCNCPoint2[23558] = {X 607.6965, Y 36.8536, Z 0.0000, A 0.000, B 0.000, C 0.000 }
gfCNCPoint2[23559] = {X 607.6965, Y 36.8536, Z -3.0000, A 0.000, B 0.000, C 0.000 }
gfCNCPoint2[23560] = {X 603.6965, Y 46.5283, Z -3.0000, A 0.000, B 0.000, C 0.000 }
gfCNCPoint2[23561] = {X 603.5430, Y 46.8566, Z -3.0000, A 0.000, B 0.000, C 0.000 }
gfCNCPoint2[23562] = {X 603.3605, Y 47.1696, Z -3.0000, A 0.000, B 0.000, C 0.000 }
gfCNCPoint2[23563] = {X 602.8638, Y 47.7926, Z -3.0000, A 0.000, B 0.000, C 0.000 }
gfCNCPoint2[23564] = {X 602.2536, Y 48.3047, Z -3.0000, A 0.000, B 0.000, C 0.000 }
gfCNCPoint2[23565] = {X 601.5540, Y 48.6858, Z -3.0000, A 0.000, B 0.000, C 0.000 }
gfCNCPoint2[23566] = {X 600.7927, Y 48.9207, Z -3.0000, A 0.000, B 0.000, C 0.000 }
gfCNCPoint2[23567] = {X 600.0000, Y 49.0000, Z -3.0000, A 0.000, B 0.000, C 0.000 }
gfCNCPoint2[23568] = {X 593.5565, Y 49.0000, Z -3.0000, A 0.000, B 0.000, C 0.000 }
gfCNCPoint2[23569] = {X 592.6664, Y 48.8997, Z -3.0000, A 0.000, B 0.000, C 0.000 }
gfCNCPoint2[23570] = {X 591.8210, Y 48.6039, Z -3.0000, A 0.000, B 0.000, C 0.000 }
gfCNCPoint2[23571] = {X 591.0626, Y 48.1273, Z -3.0000, A 0.000, B 0.000, C 0.000 }
gfCNCPoint2[23572] = {X 590.4292, Y 47.4940, Z -3.0000, A 0.000, B 0.000, C 0.000 }
gfCNCPoint2[23573] = {X 589.9527, Y 46.7355, Z -3.0000, A 0.000, B 0.000, C 0.000 }
gfCNCPoint2[23574] = {X 589.6568, Y 45.8901, Z -3.0000, A 0.000, B 0.000, C 0.000 }
gfCNCPoint2[23575] = {X 589.5565, Y 45.0000, Z -3.0000, A 0.000, B 0.000, C 0.000 }
gfCNCPoint2[23576] = {X 589.5565, Y 44.0660, Z -3.0000, A 0.000, B 0.000, C 0.000 }
gfCNCPoint2[23577] = {X 589.6616, Y 43.1706, Z -3.0000, A 0.000, B 0.000, C 0.000 }
gfCNCPoint2[23578] = {X 589.9624, Y 42.3208, Z -3.0000, A 0.000, B 0.000, C 0.000 }
gfCNCPoint2[23579] = {X 590.4441, Y 41.5587, Z -3.0000, A 0.000, B 0.000, C 0.000 }
gfCNCPoint2[23580] = {X 591.0827, Y 40.9224, Z -3.0000, A 0.000, B 0.000, C 0.000 }
gfCNCPoint2[23581] = {X 591.0833, Y 40.7358, Z -3.0000, A 0.000, B 0.000, C 0.000 }
gfCNCPoint2[23582] = {X 591.0848, Y 40.3068, Z -3.0000, A 0.000, B 0.000, C 0.000 }
gfCNCPoint2[23583] = {X 591.0832, Y 32.0428, Z -3.0000, A 0.000, B 0.000, C 0.000 }
gfCNCPoint2[23584] = {X 590.9675, Y 32.1736, Z -3.0000, A 0.000, B 0.000, C 0.000 }
gfCNCPoint2[23585] = {X 590.3129, Y 33.7892, Z -3.0000, A 0.000, B 0.000, C 0.000 }
gfCNCPoint2[23586] = {X 585.1497, Y 46.5300, Z -3.0000, A 0.000, B 0.000, C 0.000 }
gfCNCPoint2[23587] = {X 584.8073, Y 47.1805, Z -3.0000, A 0.000, B 0.000, C 0.000 }
gfCNCPoint2[23588] = {X 584.3516, Y 47.7574, Z -3.0000, A 0.000, B 0.000, C 0.000 }
gfCNCPoint2[23589] = {X 583.7980, Y 48.2411, Z -3.0000, A 0.000, B 0.000, C 0.000 }
gfCNCPoint2[23590] = {X 583.1653, Y 48.6154, Z -3.0000, A 0.000, B 0.000, C 0.000 }
gfCNCPoint2[23591] = {X 582.2878, Y 48.9121, Z -3.0000, A 0.000, B 0.000, C 0.000 }
gfCNCPoint2[23592] = {X 581.3656, Y 48.9990, Z -3.0000, A 0.000, B 0.000, C 0.000 }
gfCNCPoint2[23593] = {X 580.4480, Y 48.8715, Z -3.0000, A 0.000, B 0.000, C 0.000 }
gfCNCPoint2[23594] = {X 579.5845, Y 48.5363, Z -3.0000, A 0.000, B 0.000, C 0.000 }
gfCNCPoint2[23595] = {X 578.8212, Y 48.0115, Z -3.0000, A 0.000, B 0.000, C 0.000 }
gfCNCPoint2[23596] = {X 578.1990, Y 47.3251, Z -3.0000, A 0.000, B 0.000, C 0.000 }
gfCNCPoint2[23597] = {X 577.7515, Y 46.5141, Z -3.0000, A 0.000, B 0.000, C 0.000 }
gfCNCPoint2[23598] = {X 571.6982, Y 31.7119, Z -3.0000, A 0.000, B 0.000, C 0.000 }
gfCNCPoint2[23599] = {X 571.6986, Y 40.9224, Z -3.0000, A 0.000, B 0.000, C 0.000 }
gfCNCPoint2[23600] = {X 571.8375, Y 41.0357, Z -3.0000, A 0.000, B 0.000, C 0.000 }
gfCNCPoint2[23601] = {X 572.4236, Y 41.6622, Z -3.0000, A 0.000, B 0.000, C 0.000 }
gfCNCPoint2[23602] = {X 572.8627, Y 42.3993, Z -3.0000, A 0.000, B 0.000, C 0.000 }
gfCNCPoint2[23603] = {X 573.1344, Y 43.2130, Z -3.0000, A 0.000, B 0.000, C 0.000 }
gfCNCPoint2[23604] = {X 573.2264, Y 44.0660, Z -3.0000, A 0.000, B 0.000, C 0.000 }
gfCNCPoint2[23605] = {X 573.2264, Y 45.0000, Z -3.0000, A 0.000, B 0.000, C 0.000 }
gfCNCPoint2[23606] = {X 573.1261, Y 45.8901, Z -3.0000, A 0.000, B 0.000, C 0.000 }
gfCNCPoint2[23607] = {X 572.8303, Y 46.7355, Z -3.0000, A 0.000, B 0.000, C 0.000 }
gfCNCPoint2[23608] = {X 572.3538, Y 47.4940, Z -3.0000, A 0.000, B 0.000, C 0.000 }
gfCNCPoint2[23609] = {X 571.7204, Y 48.1273, Z -3.0000, A 0.000, B 0.000, C 0.000 }
gfCNCPoint2[23610] = {X 570.9620, Y 48.6039, Z -3.0000, A 0.000, B 0.000, C 0.000 }
gfCNCPoint2[23611] = {X 570.1165, Y 48.8997, Z -3.0000, A 0.000, B 0.000, C 0.000 }
gfCNCPoint2[23612] = {X 569.2264, Y 49.0000, Z -3.0000, A 0.000, B 0.000, C 0.000 }
gfCNCPoint2[23613] = {X 562.4443, Y 49.0000, Z -3.0000, A 0.000, B 0.000, C 0.000 }
gfCNCPoint2[23614] = {X 561.5542, Y 48.8997, Z -3.0000, A 0.000, B 0.000, C 0.000 }
gfCNCPoint2[23615] = {X 560.7088, Y 48.6039, Z -3.0000, A 0.000, B 0.000, C 0.000 }
gfCNCPoint2[23616] = {X 559.9503, Y 48.1273, Z -3.0000, A 0.000, B 0.000, C 0.000 }
gfCNCPoint2[23617] = {X 559.3170, Y 47.4940, Z -3.0000, A 0.000, B 0.000, C 0.000 }
gfCNCPoint2[23618] = {X 558.8404, Y 46.7355, Z -3.0000, A 0.000, B 0.000, C 0.000 }
gfCNCPoint2[23619] = {X 558.5446, Y 45.8901, Z -3.0000, A 0.000, B 0.000, C 0.000 }
gfCNCPoint2[23620] = {X 558.4443, Y 45.0000, Z -3.0000, A 0.000, B 0.000, C 0.000 }
gfCNCPoint2[23621] = {X 558.4443, Y 44.0660, Z -3.0000, A 0.000, B 0.000, C 0.000 }
gfCNCPoint2[23622] = {X 558.5393, Y 43.2139, Z -3.0000, A 0.000, B 0.000, C 0.000 }
gfCNCPoint2[23623] = {X 558.8121, Y 42.4011, Z -3.0000, A 0.000, B 0.000, C 0.000 }
gfCNCPoint2[23624] = {X 559.2505, Y 41.6642, Z -3.0000, A 0.000, B 0.000, C 0.000 }
gfCNCPoint2[23625] = {X 559.8346, Y 41.0366, Z -3.0000, A 0.000, B 0.000, C 0.000 }
gfCNCPoint2[23626] = {X 559.9029, Y 40.9786, Z -3.0000, A 0.000, B 0.000, C 0.000 }
gfCNCPoint2[23627] = {X 559.9724, Y 40.9222, Z -3.0000, A 0.000, B 0.000, C 0.000 }
gfCNCPoint2[23628] = {X 559.9724, Y 9.0788, Z -3.0000, A 0.000, B 0.000, C 0.000 }
gfCNCPoint2[23629] = {X 559.3301, Y 8.4444, Z -3.0000, A 0.000, B 0.000, C 0.000 }
gfCNCPoint2[23630] = {X 558.8465, Y 7.6822, Z -3.0000, A 0.000, B 0.000, C 0.000 }
gfCNCPoint2[23631] = {X 558.5461, Y 6.8309, Z -3.0000, A 0.000, B 0.000, C 0.000 }
gfCNCPoint2[23632] = {X 558.4443, Y 5.9339, Z -3.0000, A 0.000, B 0.000, C 0.000 }
gfCNCPoint2[23633] = {X 558.4443, Y 5.0000, Z -3.0000, A 0.000, B 0.000, C 0.000 }
gfCNCPoint2[23634] = {X 558.5446, Y 4.1099, Z -3.0000, A 0.000, B 0.000, C 0.000 }
gfCNCPoint2[23635] = {X 558.8404, Y 3.2645, Z -3.0000, A 0.000, B 0.000, C 0.000 }
gfCNCPoint2[23636] = {X 559.3170, Y 2.5060, Z -3.0000, A 0.000, B 0.000, C 0.000 }
gfCNCPoint2[23637] = {X 559.9503, Y 1.8727, Z -3.0000, A 0.000, B 0.000, C 0.000 }
gfCNCPoint2[23638] = {X 560.7088, Y 1.3961, Z -3.0000, A 0.000, B 0.000, C 0.000 }
gfCNCPoint2[23639] = {X 561.5542, Y 1.1003, Z -3.0000, A 0.000, B 0.000, C 0.000 }
gfCNCPoint2[23640] = {X 562.4443, Y 1.0000, Z -3.0000, A 0.000, B 0.000, C 0.000 }
gfCNCPoint2[23641] = {X 570.9376, Y 1.0000, Z -3.0000, A 0.000, B 0.000, C 0.000 }
gfCNCPoint2[23642] = {X 571.8276, Y 1.1003, Z -3.0000, A 0.000, B 0.000, C 0.000 }
gfCNCPoint2[23643] = {X 572.6731, Y 1.3961, Z -3.0000, A 0.000, B 0.000, C 0.000 }
gfCNCPoint2[23644] = {X 573.4315, Y 1.8727, Z -3.0000, A 0.000, B 0.000, C 0.000 }
gfCNCPoint2[23645] = {X 574.0649, Y 2.5060, Z -3.0000, A 0.000, B 0.000, C 0.000 }
gfCNCPoint2[23646] = {X 574.5414, Y 3.2645, Z -3.0000, A 0.000, B 0.000, C 0.000 }
gfCNCPoint2[23647] = {X 574.8373, Y 4.1099, Z -3.0000, A 0.000, B 0.000, C 0.000 }
gfCNCPoint2[23648] = {X 574.9376, Y 5.0000, Z -3.0000, A 0.000, B 0.000, C 0.000 }
gfCNCPoint2[23649] = {X 574.9372, Y 5.9858, Z -3.0000, A 0.000, B 0.000, C 0.000 }
gfCNCPoint2[23650] = {X 574.8649, Y 6.6931, Z -3.0000, A 0.000, B 0.000, C 0.000 }
gfCNCPoint2[23651] = {X 574.6685, Y 7.3763, Z -3.0000, A 0.000, B 0.000, C 0.000 }
gfCNCPoint2[23652] = {X 574.3542, Y 8.0141, Z -3.0000, A 0.000, B 0.000, C 0.000 }
gfCNCPoint2[23653] = {X 574.2917, Y 8.1134, Z -3.0000, A 0.000, B 0.000, C 0.000 }
gfCNCPoint2[23654] = {X 574.2264, Y 8.2108, Z -3.0000, A 0.000, B 0.000, C 0.000 }
gfCNCPoint2[23655] = {X 574.2610, Y 8.2363, Z -3.0000, A 0.000, B 0.000, C 0.000 }
gfCNCPoint2[23656] = {X 574.2842, Y 8.2723, Z -3.0000, A 0.000, B 0.000, C 0.000 }
gfCNCPoint2[23657] = {X 574.6456, Y 9.1532, Z -3.0000, A 0.000, B 0.000, C 0.000 }
gfCNCPoint2[23658] = {X 581.1904, Y 25.2173, Z -3.0000, A 0.000, B 0.000, C 0.000 }
gfCNCPoint2[23659] = {X 588.2029, Y 8.0668, Z -3.0000, A 0.000, B 0.000, C 0.000 }
gfCNCPoint2[23660] = {X 587.8648, Y 7.3987, Z -3.0000, A 0.000, B 0.000, C 0.000 }
gfCNCPoint2[23661] = {X 587.6570, Y 6.6794, Z -3.0000, A 0.000, B 0.000, C 0.000 }
gfCNCPoint2[23662] = {X 587.5870, Y 5.9339, Z -3.0000, A 0.000, B 0.000, C 0.000 }
gfCNCPoint2[23663] = {X 587.5870, Y 5.0000, Z -3.0000, A 0.000, B 0.000, C 0.000 }
gfCNCPoint2[23664] = {X 587.6872, Y 4.1099, Z -3.0000, A 0.000, B 0.000, C 0.000 }
gfCNCPoint2[23665] = {X 587.9831, Y 3.2645, Z -3.0000, A 0.000, B 0.000, C 0.000 }
gfCNCPoint2[23666] = {X 588.4596, Y 2.5060, Z -3.0000, A 0.000, B 0.000, C 0.000 }
gfCNCPoint2[23667] = {X 589.0930, Y 1.8727, Z -3.0000, A 0.000, B 0.000, C 0.000 }
gfCNCPoint2[23668] = {X 589.8514, Y 1.3961, Z -3.0000, A 0.000, B 0.000, C 0.000 }
gfCNCPoint2[23669] = {X 590.6969, Y 1.1003, Z -3.0000, A 0.000, B 0.000, C 0.000 }
gfCNCPoint2[23670] = {X 591.5870, Y 1.0000, Z -3.0000, A 0.000, B 0.000, C 0.000 }
gfCNCPoint2[23671] = {X 600.0000, Y 1.0000, Z -3.0000, A 0.000, B 0.000, C 0.000 }
gfCNCPoint2[23672] = {X 600.7927, Y 1.0793, Z -3.0000, A 0.000, B 0.000, C 0.000 }
gfCNCPoint2[23673] = {X 601.5540, Y 1.3142, Z -3.0000, A 0.000, B 0.000, C 0.000 }
gfCNCPoint2[23674] = {X 602.2536, Y 1.6953, Z -3.0000, A 0.000, B 0.000, C 0.000 }
gfCNCPoint2[23675] = {X 602.8638, Y 2.2074, Z -3.0000, A 0.000, B 0.000, C 0.000 }
gfCNCPoint2[23676] = {X 603.3605, Y 2.8304, Z -3.0000, A 0.000, B 0.000, C 0.000 }
gfCNCPoint2[23677] = {X 603.5430, Y 3.1434, Z -3.0000, A 0.000, B 0.000, C 0.000 }
gfCNCPoint2[23678] = {X 603.6965, Y 3.4717, Z -3.0000, A 0.000, B 0.000, C 0.000 }
gfCNCPoint2[23679] = {X 607.6965, Y 13.1464, Z -3.0000, A 0.000, B 0.000, C 0.000 }
gfCNCPoint2[23680] = {X 607.6965, Y 13.1464, Z 0.0000, A 0.000, B 0.000, C 0.000 }
gfCNCPoint2[23681] = {X 607.6965, Y 13.1464, Z 11.0000, A 0.000, B 0.000, C 0.000 }
gfCNCPoint2[23682] = {X 256.2427, Y 19.7804, Z 11.0000, A 0.000, B 0.000, C 0.000 }
gfCNCPoint2[23683] = {X 256.2427, Y 19.7804, Z 0.8333, A 0.000, B 0.000, C 0.000 }
gfCNCPoint2[23684] = {X 251.5292, Y 19.7804, Z -0.4296, A 0.000, B 0.000, C 0.000 }
gfCNCPoint2[23685] = {X 250.8346, Y 19.7912, Z -0.6158, A 0.000, B 0.000, C 0.000 }
gfCNCPoint2[23686] = {X 250.1807, Y 19.7928, Z -0.7910, A 0.000, B 0.000, C 0.000 }
gfCNCPoint2[23687] = {X 249.4957, Y 19.8911, Z -0.9764, A 0.000, B 0.000, C 0.000 }
gfCNCPoint2[23688] = {X 248.8452, Y 20.0794, Z -1.1579, A 0.000, B 0.000, C 0.000 }
gfCNCPoint2[23689] = {X 248.7081, Y 20.1106, Z -1.1956, A 0.000, B 0.000, C 0.000 }
gfCNCPoint2[23690] = {X 248.6537, Y 20.1616, Z -1.2155, A 0.000, B 0.000, C 0.000 }
gfCNCPoint2[23691] = {X 248.6137, Y 20.2964, Z -1.2532, A 0.000, B 0.000, C 0.000 }
gfCNCPoint2[23692] = {X 248.4746, Y 20.7646, Z -1.3841, A 0.000, B 0.000, C 0.000 }
gfCNCPoint2[23693] = {X 248.4446, Y 21.8679, Z -1.6798, A 0.000, B 0.000, C 0.000 }
gfCNCPoint2[23694] = {X 248.5579, Y 22.3430, Z -1.8107, A 0.000, B 0.000, C 0.000 }
gfCNCPoint2[23695] = {X 248.8721, Y 22.4374, Z -1.8986, A 0.000, B 0.000, C 0.000 }
gfCNCPoint2[23696] = {X 250.4392, Y 22.5681, Z -2.3199, A 0.000, B 0.000, C 0.000 }
gfCNCPoint2[23697] = {X 251.6873, Y 22.5560, Z -2.6544, A 0.000, B 0.000, C 0.000 }
gfCNCPoint2[23698] = {X 252.9771, Y 22.5560, Z -3.0000, A 0.000, B 0.000, C 0.000 }
gfCNCPoint2[23699] = {X 257.4115, Y 22.5560, Z -3.0000, A 0.000, B 0.000, C 0.000 }
gfCNCPoint2[23700] = {X 257.4115, Y 19.7804, Z -3.0000, A 0.000, B 0.000, C 0.000 }
gfCNCPoint2[23701] = {X 251.5292, Y 19.7804, Z -3.0000, A 0.000, B 0.000, C 0.000 }
gfCNCPoint2[23702] = {X 250.8346, Y 19.7912, Z -3.0000, A 0.000, B 0.000, C 0.000 }
gfCNCPoint2[23703] = {X 249.8297, Y 19.8647, Z -3.0000, A 0.000, B 0.000, C 0.000 }
gfCNCPoint2[23704] = {X 248.8452, Y 20.0794, Z -3.0000, A 0.000, B 0.000, C 0.000 }
gfCNCPoint2[23705] = {X 248.7000, Y 20.1566, Z -3.0000, A 0.000, B 0.000, C 0.000 }
gfCNCPoint2[23706] = {X 248.6137, Y 20.2964, Z -3.0000, A 0.000, B 0.000, C 0.000 }
gfCNCPoint2[23707] = {X 248.4757, Y 20.9719, Z -3.0000, A 0.000, B 0.000, C 0.000 }
gfCNCPoint2[23708] = {X 248.4569, Y 21.6610, Z -3.0000, A 0.000, B 0.000, C 0.000 }
gfCNCPoint2[23709] = {X 248.5579, Y 22.3430, Z -3.0000, A 0.000, B 0.000, C 0.000 }
gfCNCPoint2[23710] = {X 248.8753, Y 22.4206, Z -3.0000, A 0.000, B 0.000, C 0.000 }
gfCNCPoint2[23711] = {X 249.1991, Y 22.4647, Z -3.0000, A 0.000, B 0.000, C 0.000 }
gfCNCPoint2[23712] = {X 250.4422, Y 22.5393, Z -3.0000, A 0.000, B 0.000, C 0.000 }
gfCNCPoint2[23713] = {X 251.6873, Y 22.5560, Z -3.0000, A 0.000, B 0.000, C 0.000 }
gfCNCPoint2[23714] = {X 252.9771, Y 22.5560, Z -3.0000, A 0.000, B 0.000, C 0.000 }
gfCNCPoint2[23715] = {X 248.9923, Y 22.2874, Z -3.0000, A 0.000, B 0.000, C 0.000 }
gfCNCPoint2[23716] = {X 252.9771, Y 22.6360, Z -3.0000, A 0.000, B 0.000, C 0.000 }
gfCNCPoint2[23717] = {X 257.4915, Y 22.6360, Z -3.0000, A 0.000, B 0.000, C 0.000 }
gfCNCPoint2[23718] = {X 257.4915, Y 19.7004, Z -3.0000, A 0.000, B 0.000, C 0.000 }
gfCNCPoint2[23719] = {X 251.5286, Y 19.7004, Z -3.0000, A 0.000, B 0.000, C 0.000 }
gfCNCPoint2[23720] = {X 250.8365, Y 19.7112, Z -3.0000, A 0.000, B 0.000, C 0.000 }
gfCNCPoint2[23721] = {X 249.8259, Y 19.7847, Z -3.0000, A 0.000, B 0.000, C 0.000 }
gfCNCPoint2[23722] = {X 248.8356, Y 19.9996, Z -3.0000, A 0.000, B 0.000, C 0.000 }
gfCNCPoint2[23723] = {X 248.6484, Y 20.0953, Z -3.0000, A 0.000, B 0.000, C 0.000 }
gfCNCPoint2[23724] = {X 248.5370, Y 20.2736, Z -3.0000, A 0.000, B 0.000, C 0.000 }
gfCNCPoint2[23725] = {X 248.3945, Y 20.9779, Z -3.0000, A 0.000, B 0.000, C 0.000 }
gfCNCPoint2[23726] = {X 248.3790, Y 21.6963, Z -3.0000, A 0.000, B 0.000, C 0.000 }
gfCNCPoint2[23727] = {X 248.4910, Y 22.4061, Z -3.0000, A 0.000, B 0.000, C 0.000 }
gfCNCPoint2[23728] = {X 248.8379, Y 22.4948, Z -3.0000, A 0.000, B 0.000, C 0.000 }
gfCNCPoint2[23729] = {X 249.1925, Y 22.5444, Z -3.0000, A 0.000, B 0.000, C 0.000 }
gfCNCPoint2[23730] = {X 250.4381, Y 22.6192, Z -3.0000, A 0.000, B 0.000, C 0.000 }
gfCNCPoint2[23731] = {X 251.6858, Y 22.6360, Z -3.0000, A 0.000, B 0.000, C 0.000 }
gfCNCPoint2[23732] = {X 252.9771, Y 22.6360, Z -3.0000, A 0.000, B 0.000, C 0.000 }
gfCNCPoint2[23733] = {X 256.9619, Y 22.2874, Z -3.0000, A 0.000, B 0.000, C 0.000 }
gfCNCPoint2[23734] = {X 248.9923, Y 22.3674, Z -3.0000, A 0.000, B 0.000, C 0.000 }
gfCNCPoint2[23735] = {X 252.9771, Y 22.7160, Z -3.0000, A 0.000, B 0.000, C 0.000 }
gfCNCPoint2[23736] = {X 257.5715, Y 22.7160, Z -3.0000, A 0.000, B 0.000, C 0.000 }
gfCNCPoint2[23737] = {X 257.5715, Y 19.6204, Z -3.0000, A 0.000, B 0.000, C 0.000 }
gfCNCPoint2[23738] = {X 251.5280, Y 19.6204, Z -3.0000, A 0.000, B 0.000, C 0.000 }
gfCNCPoint2[23739] = {X 250.8358, Y 19.6312, Z -3.0000, A 0.000, B 0.000, C 0.000 }
gfCNCPoint2[23740] = {X 249.8156, Y 19.7054, Z -3.0000, A 0.000, B 0.000, C 0.000 }
gfCNCPoint2[23741] = {X 248.8160, Y 19.9219, Z -3.0000, A 0.000, B 0.000, C 0.000 }
gfCNCPoint2[23742] = {X 248.5930, Y 20.0376, Z -3.0000, A 0.000, B 0.000, C 0.000 }
gfCNCPoint2[23743] = {X 248.4603, Y 20.2509, Z -3.0000, A 0.000, B 0.000, C 0.000 }
gfCNCPoint2[23744] = {X 248.3134, Y 20.9838, Z -3.0000, A 0.000, B 0.000, C 0.000 }
gfCNCPoint2[23745] = {X 248.3013, Y 21.7313, Z -3.0000, A 0.000, B 0.000, C 0.000 }
gfCNCPoint2[23746] = {X 248.4244, Y 22.4686, Z -3.0000, A 0.000, B 0.000, C 0.000 }
gfCNCPoint2[23747] = {X 248.8005, Y 22.5689, Z -3.0000, A 0.000, B 0.000, C 0.000 }
gfCNCPoint2[23748] = {X 249.1858, Y 22.6241, Z -3.0000, A 0.000, B 0.000, C 0.000 }
gfCNCPoint2[23749] = {X 250.4349, Y 22.6991, Z -3.0000, A 0.000, B 0.000, C 0.000 }
gfCNCPoint2[23750] = {X 251.6862, Y 22.7160, Z -3.0000, A 0.000, B 0.000, C 0.000 }
gfCNCPoint2[23751] = {X 252.9771, Y 22.7160, Z -3.0000, A 0.000, B 0.000, C 0.000 }
gfCNCPoint2[23752] = {X 256.9619, Y 22.3674, Z -3.0000, A 0.000, B 0.000, C 0.000 }
gfCNCPoint2[23753] = {X 248.9923, Y 22.4474, Z -3.0000, A 0.000, B 0.000, C 0.000 }
gfCNCPoint2[23754] = {X 252.9771, Y 22.7960, Z -3.0000, A 0.000, B 0.000, C 0.000 }
gfCNCPoint2[23755] = {X 257.6515, Y 22.7960, Z -3.0000, A 0.000, B 0.000, C 0.000 }
gfCNCPoint2[23756] = {X 257.6515, Y 19.5404, Z -3.0000, A 0.000, B 0.000, C 0.000 }
gfCNCPoint2[23757] = {X 251.5274, Y 19.5404, Z -3.0000, A 0.000, B 0.000, C 0.000 }
gfCNCPoint2[23758] = {X 250.8351, Y 19.5512, Z -3.0000, A 0.000, B 0.000, C 0.000 }
gfCNCPoint2[23759] = {X 249.8053, Y 19.6260, Z -3.0000, A 0.000, B 0.000, C 0.000 }
gfCNCPoint2[23760] = {X 248.7962, Y 19.8444, Z -3.0000, A 0.000, B 0.000, C 0.000 }
gfCNCPoint2[23761] = {X 248.5375, Y 19.9799, Z -3.0000, A 0.000, B 0.000, C 0.000 }
gfCNCPoint2[23762] = {X 248.3836, Y 20.2281, Z -3.0000, A 0.000, B 0.000, C 0.000 }
gfCNCPoint2[23763] = {X 248.2323, Y 20.9896, Z -3.0000, A 0.000, B 0.000, C 0.000 }
gfCNCPoint2[23764] = {X 248.2237, Y 21.7660, Z -3.0000, A 0.000, B 0.000, C 0.000 }
gfCNCPoint2[23765] = {X 248.3582, Y 22.5307, Z -3.0000, A 0.000, B 0.000, C 0.000 }
gfCNCPoint2[23766] = {X 248.7633, Y 22.6429, Z -3.0000, A 0.000, B 0.000, C 0.000 }
gfCNCPoint2[23767] = {X 249.1792, Y 22.7039, Z -3.0000, A 0.000, B 0.000, C 0.000 }
gfCNCPoint2[23768] = {X 250.4318, Y 22.7791, Z -3.0000, A 0.000, B 0.000, C 0.000 }
gfCNCPoint2[23769] = {X 251.6866, Y 22.7960, Z -3.0000, A 0.000, B 0.000, C 0.000 }
gfCNCPoint2[23770] = {X 252.9771, Y 22.7960, Z -3.0000, A 0.000, B 0.000, C 0.000 }
gfCNCPoint2[23771] = {X 256.9619, Y 22.4474, Z -3.0000, A 0.000, B 0.000, C 0.000 }
gfCNCPoint2[23772] = {X 248.9923, Y 22.5274, Z -3.0000, A 0.000, B 0.000, C 0.000 }
gfCNCPoint2[23773] = {X 252.9771, Y 22.8760, Z -3.0000, A 0.000, B 0.000, C 0.000 }
gfCNCPoint2[23774] = {X 257.7315, Y 22.8760, Z -3.0000, A 0.000, B 0.000, C 0.000 }
gfCNCPoint2[23775] = {X 257.7315, Y 19.4604, Z -3.0000, A 0.000, B 0.000, C 0.000 }
gfCNCPoint2[23776] = {X 251.5267, Y 19.4604, Z -3.0000, A 0.000, B 0.000, C 0.000 }
gfCNCPoint2[23777] = {X 250.8344, Y 19.4712, Z -3.0000, A 0.000, B 0.000, C 0.000 }
gfCNCPoint2[23778] = {X 249.7949, Y 19.5467, Z -3.0000, A 0.000, B 0.000, C 0.000 }
gfCNCPoint2[23779] = {X 248.7763, Y 19.7669, Z -3.0000, A 0.000, B 0.000, C 0.000 }
gfCNCPoint2[23780] = {X 248.4820, Y 19.9223, Z -3.0000, A 0.000, B 0.000, C 0.000 }
gfCNCPoint2[23781] = {X 248.3069, Y 20.2053, Z -3.0000, A 0.000, B 0.000, C 0.000 }
gfCNCPoint2[23782] = {X 248.1519, Y 20.9889, Z -3.0000, A 0.000, B 0.000, C 0.000 }
gfCNCPoint2[23783] = {X 248.1453, Y 21.7876, Z -3.0000, A 0.000, B 0.000, C 0.000 }
gfCNCPoint2[23784] = {X 248.2871, Y 22.5736, Z -3.0000, A 0.000, B 0.000, C 0.000 }
gfCNCPoint2[23785] = {X 248.3058, Y 22.5971, Z -3.0000, A 0.000, B 0.000, C 0.000 }
gfCNCPoint2[23786] = {X 248.3321, Y 22.6063, Z -3.0000, A 0.000, B 0.000, C 0.000 }
gfCNCPoint2[23787] = {X 248.7468, Y 22.7212, Z -3.0000, A 0.000, B 0.000, C 0.000 }
gfCNCPoint2[23788] = {X 249.1726, Y 22.7836, Z -3.0000, A 0.000, B 0.000, C 0.000 }
gfCNCPoint2[23789] = {X 250.4287, Y 22.8590, Z -3.0000, A 0.000, B 0.000, C 0.000 }
gfCNCPoint2[23790] = {X 251.6869, Y 22.8760, Z -3.0000, A 0.000, B 0.000, C 0.000 }
gfCNCPoint2[23791] = {X 252.9771, Y 22.8760, Z -3.0000, A 0.000, B 0.000, C 0.000 }
gfCNCPoint2[23792] = {X 256.9619, Y 22.5274, Z -3.0000, A 0.000, B 0.000, C 0.000 }
gfCNCPoint2[23793] = {X 248.9923, Y 22.6074, Z -3.0000, A 0.000, B 0.000, C 0.000 }
gfCNCPoint2[23794] = {X 252.9771, Y 22.9560, Z -3.0000, A 0.000, B 0.000, C 0.000 }
gfCNCPoint2[23795] = {X 257.8115, Y 22.9560, Z -3.0000, A 0.000, B 0.000, C 0.000 }
gfCNCPoint2[23796] = {X 257.8091, Y 19.3804, Z -3.0000, A 0.000, B 0.000, C 0.000 }
gfCNCPoint2[23797] = {X 251.5261, Y 19.3804, Z -3.0000, A 0.000, B 0.000, C 0.000 }
gfCNCPoint2[23798] = {X 250.8336, Y 19.3912, Z -3.0000, A 0.000, B 0.000, C 0.000 }
gfCNCPoint2[23799] = {X 249.7844, Y 19.4674, Z -3.0000, A 0.000, B 0.000, C 0.000 }
gfCNCPoint2[23800] = {X 248.7562, Y 19.6894, Z -3.0000, A 0.000, B 0.000, C 0.000 }
gfCNCPoint2[23801] = {X 248.4264, Y 19.8648, Z -3.0000, A 0.000, B 0.000, C 0.000 }
gfCNCPoint2[23802] = {X 248.2302, Y 20.1825, Z -3.0000, A 0.000, B 0.000, C 0.000 }
gfCNCPoint2[23803] = {X 248.0718, Y 20.9862, Z -3.0000, A 0.000, B 0.000, C 0.000 }
gfCNCPoint2[23804] = {X 248.0665, Y 21.8053, Z -3.0000, A 0.000, B 0.000, C 0.000 }
gfCNCPoint2[23805] = {X 248.2144, Y 22.6109, Z -3.0000, A 0.000, B 0.000, C 0.000 }
gfCNCPoint2[23806] = {X 248.2574, Y 22.6647, Z -3.0000, A 0.000, B 0.000, C 0.000 }
gfCNCPoint2[23807] = {X 248.7051, Y 22.7940, Z -3.0000, A 0.000, B 0.000, C 0.000 }
gfCNCPoint2[23808] = {X 249.1659, Y 22.8633, Z -3.0000, A 0.000, B 0.000, C 0.000 }
gfCNCPoint2[23809] = {X 250.4255, Y 22.9390, Z -3.0000, A 0.000, B 0.000, C 0.000 }
gfCNCPoint2[23810] = {X 251.6873, Y 22.9560, Z -3.0000, A 0.000, B 0.000, C 0.000 }
gfCNCPoint2[23811] = {X 252.9771, Y 22.9560, Z -3.0000, A 0.000, B 0.000, C 0.000 }
gfCNCPoint2[23812] = {X 256.9619, Y 22.6074, Z -3.0000, A 0.000, B 0.000, C 0.000 }
gfCNCPoint2[23813] = {X 256.9619, Y 22.6074, Z 0.0000, A 0.000, B 0.000, C 0.000 }
gfCNCPoint2[23814] = {X 256.9619, Y 22.6074, Z 11.0000, A 0.000, B 0.000, C 0.000 }
gfCNCPoint2[23815] = {X 188.4952, Y 19.4656, Z 11.0000, A 0.000, B 0.000, C 0.000 }
gfCNCPoint2[23816] = {X 188.4952, Y 19.4656, Z 0.8333, A 0.000, B 0.000, C 0.000 }
gfCNCPoint2[23817] = {X 188.3884, Y 19.4278, Z 0.8030, A 0.000, B 0.000, C 0.000 }
gfCNCPoint2[23818] = {X 187.7714, Y 19.3592, Z 0.6367, A 0.000, B 0.000, C 0.000 }
gfCNCPoint2[23819] = {X 186.9109, Y 19.2593, Z 0.4045, A 0.000, B 0.000, C 0.000 }
gfCNCPoint2[23820] = {X 184.5930, Y 19.3668, Z -0.2172, A 0.000, B 0.000, C 0.000 }
gfCNCPoint2[23821] = {X 183.7430, Y 19.5465, Z -0.4500, A 0.000, B 0.000, C 0.000 }
gfCNCPoint2[23822] = {X 183.0414, Y 19.6903, Z -0.6419, A 0.000, B 0.000, C 0.000 }
gfCNCPoint2[23823] = {X 182.0255, Y 20.0600, Z -0.9316, A 0.000, B 0.000, C 0.000 }
gfCNCPoint2[23824] = {X 181.3956, Y 20.4009, Z -1.1235, A 0.000, B 0.000, C 0.000 }
gfCNCPoint2[23825] = {X 181.3397, Y 20.9125, Z -1.2614, A 0.000, B 0.000, C 0.000 }
gfCNCPoint2[23826] = {X 180.8643, Y 22.1272, Z -1.6109, A 0.000, B 0.000, C 0.000 }
gfCNCPoint2[23827] = {X 180.5581, Y 22.5409, Z -1.7488, A 0.000, B 0.000, C 0.000 }
gfCNCPoint2[23828] = {X 182.2908, Y 22.3349, Z -2.2164, A 0.000, B 0.000, C 0.000 }
gfCNCPoint2[23829] = {X 182.5945, Y 22.3103, Z -2.2980, A 0.000, B 0.000, C 0.000 }
gfCNCPoint2[23830] = {X 184.3414, Y 22.2341, Z -2.7666, A 0.000, B 0.000, C 0.000 }
gfCNCPoint2[23831] = {X 184.7767, Y 22.2191, Z -2.8833, A 0.000, B 0.000, C 0.000 }
gfCNCPoint2[23832] = {X 185.2119, Y 22.2007, Z -3.0000, A 0.000, B 0.000, C 0.000 }
gfCNCPoint2[23833] = {X 187.5426, Y 22.0781, Z -3.0000, A 0.000, B 0.000, C 0.000 }
gfCNCPoint2[23834] = {X 189.8702, Y 21.9075, Z -3.0000, A 0.000, B 0.000, C 0.000 }
gfCNCPoint2[23835] = {X 190.4718, Y 21.8316, Z -3.0000, A 0.000, B 0.000, C 0.000 }
gfCNCPoint2[23836] = {X 191.0591, Y 21.6802, Z -3.0000, A 0.000, B 0.000, C 0.000 }
gfCNCPoint2[23837] = {X 191.0689, Y 21.1640, Z -3.0000, A 0.000, B 0.000, C 0.000 }
gfCNCPoint2[23838] = {X 190.8730, Y 20.6863, Z -3.0000, A 0.000, B 0.000, C 0.000 }
gfCNCPoint2[23839] = {X 190.5036, Y 20.3256, Z -3.0000, A 0.000, B 0.000, C 0.000 }
gfCNCPoint2[23840] = {X 189.6460, Y 19.8647, Z -3.0000, A 0.000, B 0.000, C 0.000 }
gfCNCPoint2[23841] = {X 188.7281, Y 19.5401, Z -3.0000, A 0.000, B 0.000, C 0.000 }
gfCNCPoint2[23842] = {X 187.7714, Y 19.3592, Z -3.0000, A 0.000, B 0.000, C 0.000 }
gfCNCPoint2[23843] = {X 186.4245, Y 19.2761, Z -3.0000, A 0.000, B 0.000, C 0.000 }
gfCNCPoint2[23844] = {X 185.0764, Y 19.3388, Z -3.0000, A 0.000, B 0.000, C 0.000 }
gfCNCPoint2[23845] = {X 183.7430, Y 19.5465, Z -3.0000, A 0.000, B 0.000, C 0.000 }
gfCNCPoint2[23846] = {X 182.5379, Y 19.8873, Z -3.0000, A 0.000, B 0.000, C 0.000 }
gfCNCPoint2[23847] = {X 181.3956, Y 20.4009, Z -3.0000, A 0.000, B 0.000, C 0.000 }
gfCNCPoint2[23848] = {X 181.2442, Y 21.1599, Z -3.0000, A 0.000, B 0.000, C 0.000 }
gfCNCPoint2[23849] = {X 180.9621, Y 21.8807, Z -3.0000, A 0.000, B 0.000, C 0.000 }
gfCNCPoint2[23850] = {X 180.5581, Y 22.5409, Z -3.0000, A 0.000, B 0.000, C 0.000 }
gfCNCPoint2[23851] = {X 182.4469, Y 22.3521, Z -3.0000, A 0.000, B 0.000, C 0.000 }
gfCNCPoint2[23852] = {X 184.3414, Y 22.2341, Z -3.0000, A 0.000, B 0.000, C 0.000 }
gfCNCPoint2[23853] = {X 184.7767, Y 22.2183, Z -3.0000, A 0.000, B 0.000, C 0.000 }
gfCNCPoint2[23854] = {X 185.2119, Y 22.2007, Z -3.0000, A 0.000, B 0.000, C 0.000 }
gfCNCPoint2[23855] = {X 181.2194, Y 22.1006, Z -3.0000, A 0.000, B 0.000, C 0.000 }
gfCNCPoint2[23856] = {X 185.2153, Y 22.2806, Z -3.0000, A 0.000, B 0.000, C 0.000 }
gfCNCPoint2[23857] = {X 187.5451, Y 22.1581, Z -3.0000, A 0.000, B 0.000, C 0.000 }
gfCNCPoint2[23858] = {X 189.8718, Y 21.9876, Z -3.0000, A 0.000, B 0.000, C 0.000 }
gfCNCPoint2[23859] = {X 190.5071, Y 21.9062, Z -3.0000, A 0.000, B 0.000, C 0.000 }
gfCNCPoint2[23860] = {X 191.1263, Y 21.7422, Z -3.0000, A 0.000, B 0.000, C 0.000 }
gfCNCPoint2[23861] = {X 191.1528, Y 21.1792, Z -3.0000, A 0.000, B 0.000, C 0.000 }
gfCNCPoint2[23862] = {X 190.9478, Y 20.6542, Z -3.0000, A 0.000, B 0.000, C 0.000 }
gfCNCPoint2[23863] = {X 190.5468, Y 20.2582, Z -3.0000, A 0.000, B 0.000, C 0.000 }
gfCNCPoint2[23864] = {X 189.6790, Y 19.7919, Z -3.0000, A 0.000, B 0.000, C 0.000 }
gfCNCPoint2[23865] = {X 188.7502, Y 19.4632, Z -3.0000, A 0.000, B 0.000, C 0.000 }
gfCNCPoint2[23866] = {X 187.7823, Y 19.2800, Z -3.0000, A 0.000, B 0.000, C 0.000 }
gfCNCPoint2[23867] = {X 186.4270, Y 19.1961, Z -3.0000, A 0.000, B 0.000, C 0.000 }
gfCNCPoint2[23868] = {X 185.0706, Y 19.2590, Z -3.0000, A 0.000, B 0.000, C 0.000 }
gfCNCPoint2[23869] = {X 183.7289, Y 19.4677, Z -3.0000, A 0.000, B 0.000, C 0.000 }
gfCNCPoint2[23870] = {X 182.4922, Y 19.8188, Z -3.0000, A 0.000, B 0.000, C 0.000 }
gfCNCPoint2[23871] = {X 181.3216, Y 20.3500, Z -3.0000, A 0.000, B 0.000, C 0.000 }
gfCNCPoint2[23872] = {X 181.1582, Y 21.1711, Z -3.0000, A 0.000, B 0.000, C 0.000 }
gfCNCPoint2[23873] = {X 180.8395, Y 21.9452, Z -3.0000, A 0.000, B 0.000, C 0.000 }
gfCNCPoint2[23874] = {X 180.3776, Y 22.6433, Z -3.0000, A 0.000, B 0.000, C 0.000 }
gfCNCPoint2[23875] = {X 182.3569, Y 22.4398, Z -3.0000, A 0.000, B 0.000, C 0.000 }
gfCNCPoint2[23876] = {X 184.3427, Y 22.3141, Z -3.0000, A 0.000, B 0.000, C 0.000 }
gfCNCPoint2[23877] = {X 184.7790, Y 22.2982, Z -3.0000, A 0.000, B 0.000, C 0.000 }
gfCNCPoint2[23878] = {X 185.2153, Y 22.2806, Z -3.0000, A 0.000, B 0.000, C 0.000 }
gfCNCPoint2[23879] = {X 189.1818, Y 21.7640, Z -3.0000, A 0.000, B 0.000, C 0.000 }
gfCNCPoint2[23880] = {X 181.2227, Y 22.1805, Z -3.0000, A 0.000, B 0.000, C 0.000 }
gfCNCPoint2[23881] = {X 185.2187, Y 22.3606, Z -3.0000, A 0.000, B 0.000, C 0.000 }
gfCNCPoint2[23882] = {X 187.5497, Y 22.2380, Z -3.0000, A 0.000, B 0.000, C 0.000 }
gfCNCPoint2[23883] = {X 189.8776, Y 22.0674, Z -3.0000, A 0.000, B 0.000, C 0.000 }
gfCNCPoint2[23884] = {X 190.5438, Y 21.9805, Z -3.0000, A 0.000, B 0.000, C 0.000 }
gfCNCPoint2[23885] = {X 191.1920, Y 21.8043, Z -3.0000, A 0.000, B 0.000, C 0.000 }
gfCNCPoint2[23886] = {X 191.2497, Y 21.3481, Z -3.0000, A 0.000, B 0.000, C 0.000 }
gfCNCPoint2[23887] = {X 191.1601, Y 20.8971, Z -3.0000, A 0.000, B 0.000, C 0.000 }
gfCNCPoint2[23888] = {X 190.9324, Y 20.4977, Z -3.0000, A 0.000, B 0.000, C 0.000 }
gfCNCPoint2[23889] = {X 190.5899, Y 20.1908, Z -3.0000, A 0.000, B 0.000, C 0.000 }
gfCNCPoint2[23890] = {X 189.7113, Y 19.7187, Z -3.0000, A 0.000, B 0.000, C 0.000 }
gfCNCPoint2[23891] = {X 188.7711, Y 19.3860, Z -3.0000, A 0.000, B 0.000, C 0.000 }
gfCNCPoint2[23892] = {X 187.7911, Y 19.2004, Z -3.0000, A 0.000, B 0.000, C 0.000 }
gfCNCPoint2[23893] = {X 186.4273, Y 19.1161, Z -3.0000, A 0.000, B 0.000, C 0.000 }
gfCNCPoint2[23894] = {X 185.0625, Y 19.1794, Z -3.0000, A 0.000, B 0.000, C 0.000 }
gfCNCPoint2[23895] = {X 183.7123, Y 19.3894, Z -3.0000, A 0.000, B 0.000, C 0.000 }
gfCNCPoint2[23896] = {X 182.4466, Y 19.7503, Z -3.0000, A 0.000, B 0.000, C 0.000 }
gfCNCPoint2[23897] = {X 181.2498, Y 20.2982, Z -3.0000, A 0.000, B 0.000, C 0.000 }
gfCNCPoint2[23898] = {X 181.2398, Y 20.3522, Z -3.0000, A 0.000, B 0.000, C 0.000 }
gfCNCPoint2[23899] = {X 181.0789, Y 21.1543, Z -3.0000, A 0.000, B 0.000, C 0.000 }
gfCNCPoint2[23900] = {X 180.7669, Y 21.9106, Z -3.0000, A 0.000, B 0.000, C 0.000 }
gfCNCPoint2[23901] = {X 180.3154, Y 22.5929, Z -3.0000, A 0.000, B 0.000, C 0.000 }
gfCNCPoint2[23902] = {X 180.2507, Y 22.6709, Z -3.0000, A 0.000, B 0.000, C 0.000 }
gfCNCPoint2[23903] = {X 180.1841, Y 22.7473, Z -3.0000, A 0.000, B 0.000, C 0.000 }
gfCNCPoint2[23904] = {X 180.1888, Y 22.7475, Z -3.0000, A 0.000, B 0.000, C 0.000 }
gfCNCPoint2[23905] = {X 180.2881, Y 22.7350, Z -3.0000, A 0.000, B 0.000, C 0.000 }
gfCNCPoint2[23906] = {X 180.3873, Y 22.7227, Z -3.0000, A 0.000, B 0.000, C 0.000 }
gfCNCPoint2[23907] = {X 182.3633, Y 22.5195, Z -3.0000, A 0.000, B 0.000, C 0.000 }
gfCNCPoint2[23908] = {X 184.3458, Y 22.3941, Z -3.0000, A 0.000, B 0.000, C 0.000 }
gfCNCPoint2[23909] = {X 184.7823, Y 22.3782, Z -3.0000, A 0.000, B 0.000, C 0.000 }
gfCNCPoint2[23910] = {X 185.2187, Y 22.3606, Z -3.0000, A 0.000, B 0.000, C 0.000 }
gfCNCPoint2[23911] = {X 189.1852, Y 21.8440, Z -3.0000, A 0.000, B 0.000, C 0.000 }
gfCNCPoint2[23912] = {X 181.2261, Y 22.2605, Z -3.0000, A 0.000, B 0.000, C 0.000 }
gfCNCPoint2[23913] = {X 185.2221, Y 22.4405, Z -3.0000, A 0.000, B 0.000, C 0.000 }
gfCNCPoint2[23914] = {X 187.5543, Y 22.3178, Z -3.0000, A 0.000, B 0.000, C 0.000 }
gfCNCPoint2[23915] = {X 189.8834, Y 22.1472, Z -3.0000, A 0.000, B 0.000, C 0.000 }
gfCNCPoint2[23916] = {X 190.5798, Y 22.0549, Z -3.0000, A 0.000, B 0.000, C 0.000 }
gfCNCPoint2[23917] = {X 191.2565, Y 21.8664, Z -3.0000, A 0.000, B 0.000, C 0.000 }
gfCNCPoint2[23918] = {X 191.3305, Y 21.3763, Z -3.0000, A 0.000, B 0.000, C 0.000 }
gfCNCPoint2[23919] = {X 191.2422, Y 20.8886, Z -3.0000, A 0.000, B 0.000, C 0.000 }
gfCNCPoint2[23920] = {X 191.0011, Y 20.4555, Z -3.0000, A 0.000, B 0.000, C 0.000 }
gfCNCPoint2[23921] = {X 190.6331, Y 20.1234, Z -3.0000, A 0.000, B 0.000, C 0.000 }
gfCNCPoint2[23922] = {X 189.7437, Y 19.6455, Z -3.0000, A 0.000, B 0.000, C 0.000 }
gfCNCPoint2[23923] = {X 188.7919, Y 19.3088, Z -3.0000, A 0.000, B 0.000, C 0.000 }
gfCNCPoint2[23924] = {X 187.7999, Y 19.1209, Z -3.0000, A 0.000, B 0.000, C 0.000 }
gfCNCPoint2[23925] = {X 186.4277, Y 19.0361, Z -3.0000, A 0.000, B 0.000, C 0.000 }
gfCNCPoint2[23926] = {X 185.0543, Y 19.0998, Z -3.0000, A 0.000, B 0.000, C 0.000 }
gfCNCPoint2[23927] = {X 183.6958, Y 19.3111, Z -3.0000, A 0.000, B 0.000, C 0.000 }
gfCNCPoint2[23928] = {X 182.4009, Y 19.6820, Z -3.0000, A 0.000, B 0.000, C 0.000 }
gfCNCPoint2[23929] = {X 181.1780, Y 20.2466, Z -3.0000, A 0.000, B 0.000, C 0.000 }
gfCNCPoint2[23930] = {X 181.1605, Y 20.3408, Z -3.0000, A 0.000, B 0.000, C 0.000 }
gfCNCPoint2[23931] = {X 180.9651, Y 21.2476, Z -3.0000, A 0.000, B 0.000, C 0.000 }
gfCNCPoint2[23932] = {X 180.5735, Y 22.0885, Z -3.0000, A 0.000, B 0.000, C 0.000 }
gfCNCPoint2[23933] = {X 180.0054, Y 22.8218, Z -3.0000, A 0.000, B 0.000, C 0.000 }
gfCNCPoint2[23934] = {X 180.1926, Y 22.8276, Z -3.0000, A 0.000, B 0.000, C 0.000 }
gfCNCPoint2[23935] = {X 182.2671, Y 22.6079, Z -3.0000, A 0.000, B 0.000, C 0.000 }
gfCNCPoint2[23936] = {X 184.3489, Y 22.4740, Z -3.0000, A 0.000, B 0.000, C 0.000 }
gfCNCPoint2[23937] = {X 184.7855, Y 22.4581, Z -3.0000, A 0.000, B 0.000, C 0.000 }
gfCNCPoint2[23938] = {X 185.2221, Y 22.4405, Z -3.0000, A 0.000, B 0.000, C 0.000 }
gfCNCPoint2[23939] = {X 189.1886, Y 21.9239, Z -3.0000, A 0.000, B 0.000, C 0.000 }
gfCNCPoint2[23940] = {X 181.2295, Y 22.3404, Z -3.0000, A 0.000, B 0.000, C 0.000 }
gfCNCPoint2[23941] = {X 185.2255, Y 22.5204, Z -3.0000, A 0.000, B 0.000, C 0.000 }
gfCNCPoint2[23942] = {X 187.5589, Y 22.3977, Z -3.0000, A 0.000, B 0.000, C 0.000 }
gfCNCPoint2[23943] = {X 189.8892, Y 22.2270, Z -3.0000, A 0.000, B 0.000, C 0.000 }
gfCNCPoint2[23944] = {X 190.6153, Y 22.1292, Z -3.0000, A 0.000, B 0.000, C 0.000 }
gfCNCPoint2[23945] = {X 191.3199, Y 21.9287, Z -3.0000, A 0.000, B 0.000, C 0.000 }
gfCNCPoint2[23946] = {X 191.4106, Y 21.4048, Z -3.0000, A 0.000, B 0.000, C 0.000 }
gfCNCPoint2[23947] = {X 191.3241, Y 20.8803, Z -3.0000, A 0.000, B 0.000, C 0.000 }
gfCNCPoint2[23948] = {X 191.0698, Y 20.4134, Z -3.0000, A 0.000, B 0.000, C 0.000 }
gfCNCPoint2[23949] = {X 190.6762, Y 20.0561, Z -3.0000, A 0.000, B 0.000, C 0.000 }
gfCNCPoint2[23950] = {X 189.7761, Y 19.5724, Z -3.0000, A 0.000, B 0.000, C 0.000 }
gfCNCPoint2[23951] = {X 188.8128, Y 19.2315, Z -3.0000, A 0.000, B 0.000, C 0.000 }
gfCNCPoint2[23952] = {X 187.8088, Y 19.0414, Z -3.0000, A 0.000, B 0.000, C 0.000 }
gfCNCPoint2[23953] = {X 186.4280, Y 18.9561, Z -3.0000, A 0.000, B 0.000, C 0.000 }
gfCNCPoint2[23954] = {X 185.0462, Y 19.0202, Z -3.0000, A 0.000, B 0.000, C 0.000 }
gfCNCPoint2[23955] = {X 183.6792, Y 19.2329, Z -3.0000, A 0.000, B 0.000, C 0.000 }
gfCNCPoint2[23956] = {X 182.3552, Y 19.6136, Z -3.0000, A 0.000, B 0.000, C 0.000 }
gfCNCPoint2[23957] = {X 181.1062, Y 20.1952, Z -3.0000, A 0.000, B 0.000, C 0.000 }
gfCNCPoint2[23958] = {X 181.0813, Y 20.3295, Z -3.0000, A 0.000, B 0.000, C 0.000 }
gfCNCPoint2[23959] = {X 180.8699, Y 21.2784, Z -3.0000, A 0.000, B 0.000, C 0.000 }
gfCNCPoint2[23960] = {X 180.4400, Y 22.1504, Z -3.0000, A 0.000, B 0.000, C 0.000 }
gfCNCPoint2[23961] = {X 179.8160, Y 22.8959, Z -3.0000, A 0.000, B 0.000, C 0.000 }
gfCNCPoint2[23962] = {X 180.1965, Y 22.9078, Z -3.0000, A 0.000, B 0.000, C 0.000 }
gfCNCPoint2[23963] = {X 182.2706, Y 22.6879, Z -3.0000, A 0.000, B 0.000, C 0.000 }
gfCNCPoint2[23964] = {X 184.3521, Y 22.5540, Z -3.0000, A 0.000, B 0.000, C 0.000 }
gfCNCPoint2[23965] = {X 184.7888, Y 22.5380, Z -3.0000, A 0.000, B 0.000, C 0.000 }
gfCNCPoint2[23966] = {X 185.2255, Y 22.5204, Z -3.0000, A 0.000, B 0.000, C 0.000 }
gfCNCPoint2[23967] = {X 189.1920, Y 22.0038, Z -3.0000, A 0.000, B 0.000, C 0.000 }
gfCNCPoint2[23968] = {X 185.1538, Y 22.6035, Z -3.0000, A 0.000, B 0.000, C 0.000 }
gfCNCPoint2[23969] = {X 185.2288, Y 22.6003, Z -3.0000, A 0.000, B 0.000, C 0.000 }
gfCNCPoint2[23970] = {X 187.5635, Y 22.4776, Z -3.0000, A 0.000, B 0.000, C 0.000 }
gfCNCPoint2[23971] = {X 189.8950, Y 22.3067, Z -3.0000, A 0.000, B 0.000, C 0.000 }
gfCNCPoint2[23972] = {X 190.6503, Y 22.2036, Z -3.0000, A 0.000, B 0.000, C 0.000 }
gfCNCPoint2[23973] = {X 191.3823, Y 21.9909, Z -3.0000, A 0.000, B 0.000, C 0.000 }
gfCNCPoint2[23974] = {X 191.4903, Y 21.4336, Z -3.0000, A 0.000, B 0.000, C 0.000 }
gfCNCPoint2[23975] = {X 191.4058, Y 20.8723, Z -3.0000, A 0.000, B 0.000, C 0.000 }
gfCNCPoint2[23976] = {X 191.1386, Y 20.3715, Z -3.0000, A 0.000, B 0.000, C 0.000 }
gfCNCPoint2[23977] = {X 190.7193, Y 19.9887, Z -3.0000, A 0.000, B 0.000, C 0.000 }
gfCNCPoint2[23978] = {X 189.8085, Y 19.4992, Z -3.0000, A 0.000, B 0.000, C 0.000 }
gfCNCPoint2[23979] = {X 188.8336, Y 19.1543, Z -3.0000, A 0.000, B 0.000, C 0.000 }
gfCNCPoint2[23980] = {X 187.8176, Y 18.9619, Z -3.0000, A 0.000, B 0.000, C 0.000 }
gfCNCPoint2[23981] = {X 186.4284, Y 18.8761, Z -3.0000, A 0.000, B 0.000, C 0.000 }
gfCNCPoint2[23982] = {X 185.0380, Y 18.9406, Z -3.0000, A 0.000, B 0.000, C 0.000 }
gfCNCPoint2[23983] = {X 183.6627, Y 19.1546, Z -3.0000, A 0.000, B 0.000, C 0.000 }
gfCNCPoint2[23984] = {X 182.3094, Y 19.5454, Z -3.0000, A 0.000, B 0.000, C 0.000 }
gfCNCPoint2[23985] = {X 181.0343, Y 20.1439, Z -3.0000, A 0.000, B 0.000, C 0.000 }
gfCNCPoint2[23986] = {X 181.0020, Y 20.3183, Z -3.0000, A 0.000, B 0.000, C 0.000 }
gfCNCPoint2[23987] = {X 180.8538, Y 21.0695, Z -3.0000, A 0.000, B 0.000, C 0.000 }
gfCNCPoint2[23988] = {X 180.5651, Y 21.7787, Z -3.0000, A 0.000, B 0.000, C 0.000 }
